LIN {X -0.311,Y -646.142,Z 1277.328,A 0.000,B 0.000,C 90.000,E1 95.049} C_DIS
LIN {X -0.193,Y -640.518,Z 1277.324,A 0.000,B 0.000,C 90.000,E1 94.416} C_DIS
LIN {X 0.051,Y -635.650,Z 1277.322,A 0.000,B 0.000,C 90.000,E1 93.898} C_DIS
LIN {X -0.083,Y -629.590,Z 1277.318,A 0.000,B 0.000,C 90.000,E1 93.326} C_DIS
LIN {X -0.028,Y -623.101,Z 1277.315,A 0.000,B 0.000,C 90.000,E1 92.751} C_DIS
LIN {X 0.105,Y -616.171,Z 1277.312,A 0.000,B 0.000,C 90.000,E1 92.178} C_DIS
LIN {X -0.112,Y -607.322,Z 1277.309,A 0.000,B 0.000,C 90.000,E1 91.547} C_DIS
LIN {X -0.177,Y -601.123,Z 1277.306,A 0.000,B 0.000,C 90.000,E1 91.146} C_DIS
LIN {X 0.025,Y -594.809,Z 1277.304,A 0.000,B 0.000,C 90.000,E1 90.745} C_DIS
LIN {X 0.026,Y -587.877,Z 1277.302,A 0.000,B 0.000,C 90.000,E1 90.401} C_DIS
LIN {X -0.076,Y -580.661,Z 1277.301,A 0.000,B 0.000,C 90.000,E1 90.115} C_DIS
LIN {X 0.222,Y -575.677,Z 1277.300,A 0.000,B 0.000,C 90.000,E1 89.885} C_DIS
LIN {X -0.112,Y -572.688,Z 1277.299,A 0.000,B 0.000,C 90.000,E1 89.771} C_DIS
LIN {X 0.053,Y -572.048,Z 1277.298,A 0.000,B 0.000,C 90.000,E1 89.714} C_DIS
LIN {X -0.053,Y -569.686,Z 1277.297,A 0.000,B 0.000,C 90.000,E1 89.484} C_DIS
LIN {X 0.150,Y -569.196,Z 1277.296,A 0.000,B 0.000,C 90.000,E1 89.312} C_DIS
LIN {X -0.165,Y -568.849,Z 1277.293,A 0.000,B 0.000,C 90.000,E1 88.797} C_DIS
LIN {X -0.001,Y -570.946,Z 1277.278,A 0.000,B 0.000,C 90.000,E1 86.045} C_DIS
LIN {X -0.120,Y -572.846,Z 1277.267,A 0.000,B 0.000,C 90.000,E1 84.147} C_DIS
LIN {X 0.124,Y -574.397,Z 1277.260,A 0.000,B 0.000,C 90.000,E1 82.761} C_DIS
LIN {X 0.031,Y -576.292,Z 1277.251,A 0.000,B 0.000,C 90.000,E1 81.141} C_DIS
LIN {X -0.146,Y -577.751,Z 1277.243,A 0.000,B 0.000,C 90.000,E1 79.803} C_DIS
LIN {X -0.303,Y -578.962,Z 1277.236,A 0.000,B 0.000,C 90.000,E1 78.465} C_DIS
LIN {X 0.237,Y -580.132,Z 1277.228,A 0.000,B 0.000,C 90.000,E1 77.061} C_DIS
LIN {X -0.198,Y -581.224,Z 1277.221,A 0.000,B 0.000,C 90.000,E1 75.755} C_DIS
LIN {X 0.293,Y -581.995,Z 1277.215,A 0.000,B 0.000,C 90.000,E1 74.629} C_DIS
LIN {X 0.231,Y -582.699,Z 1277.209,A 0.000,B 0.000,C 90.000,E1 73.559} C_DIS
LIN {X 0.143,Y -584.243,Z 1277.195,A 0.000,B 0.000,C 90.000,E1 71.148} C_DIS
LIN {X 0.214,Y -585.172,Z 1277.185,A 0.000,B 0.000,C 90.000,E1 69.263} C_DIS
LIN {X -0.156,Y -586.471,Z 1277.173,A 0.000,B 0.000,C 90.000,E1 67.155} C_DIS
LIN {X -0.026,Y -587.736,Z 1277.164,A 0.000,B 0.000,C 90.000,E1 65.537} C_DIS
LIN {X -0.165,Y -588.956,Z 1277.155,A 0.000,B 0.000,C 90.000,E1 63.948} C_DIS
LIN {X -0.113,Y -590.551,Z 1277.145,A 0.000,B 0.000,C 90.000,E1 62.076} C_DIS
LIN {X 0.172,Y -591.848,Z 1277.137,A 0.000,B 0.000,C 90.000,E1 60.717} C_DIS
LIN {X 0.153,Y -593.488,Z 1277.129,A 0.000,B 0.000,C 90.000,E1 59.125} C_DIS
LIN {X 0.262,Y -594.894,Z 1277.121,A 0.000,B 0.000,C 90.000,E1 57.788} C_DIS
LIN {X 0.002,Y -596.798,Z 1277.111,A 0.000,B 0.000,C 90.000,E1 55.960} C_DIS
LIN {X -0.274,Y -598.355,Z 1277.102,A 0.000,B 0.000,C 90.000,E1 54.402} C_DIS
LIN {X 0.327,Y -599.696,Z 1277.093,A 0.000,B 0.000,C 90.000,E1 52.763} C_DIS
LIN {X -0.124,Y -601.169,Z 1277.083,A 0.000,B 0.000,C 90.000,E1 50.964} C_DIS
LIN {X 0.146,Y -601.685,Z 1277.079,A 0.000,B 0.000,C 90.000,E1 50.150} C_DIS
LIN {X -0.038,Y -602.063,Z 1277.074,A 0.000,B 0.000,C 90.000,E1 49.380} C_DIS
LIN {X 0.064,Y -602.737,Z 1277.066,A 0.000,B 0.000,C 90.000,E1 47.796} C_DIS
LIN {X 0.102,Y -603.120,Z 1277.060,A 0.000,B 0.000,C 90.000,E1 46.743} C_DIS
LIN {X -0.264,Y -603.339,Z 1277.054,A 0.000,B 0.000,C 90.000,E1 45.729} C_DIS
LIN {X 0.014,Y -603.317,Z 1277.047,A 0.000,B 0.000,C 90.000,E1 44.393} C_DIS
LIN {X -0.121,Y -603.052,Z 1277.039,A 0.000,B 0.000,C 90.000,E1 43.095} C_DIS
LIN {X 0.160,Y -602.625,Z 1277.032,A 0.000,B 0.000,C 90.000,E1 41.757} C_DIS
LIN {X 0.236,Y -602.215,Z 1277.026,A 0.000,B 0.000,C 90.000,E1 40.701} C_DIS
LIN {X 0.306,Y -601.680,Z 1277.021,A 0.000,B 0.000,C 90.000,E1 39.644} C_DIS
LIN {X -0.262,Y -601.275,Z 1277.016,A 0.000,B 0.000,C 90.000,E1 38.910} C_DIS
LIN {X 0.259,Y -600.534,Z 1277.010,A 0.000,B 0.000,C 90.000,E1 37.810} C_DIS
LIN {X 0.157,Y -599.777,Z 1277.006,A 0.000,B 0.000,C 90.000,E1 37.030} C_DIS
LIN {X 0.048,Y -598.125,Z 1276.999,A 0.000,B 0.000,C 90.000,E1 35.724} C_DIS
LIN {X -0.081,Y -596.974,Z 1276.994,A 0.000,B 0.000,C 90.000,E1 34.945} C_DIS
LIN {X 0.160,Y -595.065,Z 1276.988,A 0.000,B 0.000,C 90.000,E1 33.865} C_DIS
LIN {X -0.003,Y -593.584,Z 1276.984,A 0.000,B 0.000,C 90.000,E1 33.086} C_DIS
LIN {X 0.196,Y -590.897,Z 1276.978,A 0.000,B 0.000,C 90.000,E1 32.005} C_DIS
LIN {X 0.168,Y -588.726,Z 1276.974,A 0.000,B 0.000,C 90.000,E1 31.209} C_DIS
LIN {X 0.121,Y -586.110,Z 1276.969,A 0.000,B 0.000,C 90.000,E1 30.413} C_DIS
LIN {X 0.173,Y -584.179,Z 1276.966,A 0.000,B 0.000,C 90.000,E1 29.873} C_DIS
LIN {X 0.207,Y -581.993,Z 1276.963,A 0.000,B 0.000,C 90.000,E1 29.333} C_DIS
LIN {X 0.011,Y -577.776,Z 1276.958,A 0.000,B 0.000,C 90.000,E1 28.409} C_DIS
LIN {X -0.208,Y -575.700,Z 1276.956,A 0.000,B 0.000,C 90.000,E1 28.025} C_DIS
LIN {X 0.018,Y -570.604,Z 1276.950,A 0.000,B 0.000,C 90.000,E1 27.052} C_DIS
LIN {X 0.012,Y -565.575,Z 1276.946,A 0.000,B 0.000,C 90.000,E1 26.232} C_DIS
LIN {X 0.150,Y -562.014,Z 1276.943,A 0.000,B 0.000,C 90.000,E1 25.668} C_DIS
LIN {X -0.240,Y -558.197,Z 1276.940,A 0.000,B 0.000,C 90.000,E1 25.155} C_DIS
LIN {X -0.150,Y -554.156,Z 1276.937,A 0.000,B 0.000,C 90.000,E1 24.591} C_DIS
LIN {X -0.202,Y -548.717,Z 1276.933,A 0.000,B 0.000,C 90.000,E1 23.898} C_DIS
LIN {X -0.233,Y -541.795,Z 1276.928,A 0.000,B 0.000,C 90.000,E1 23.078} C_DIS
LIN {X 0.234,Y -536.783,Z 1276.925,A 0.000,B 0.000,C 90.000,E1 22.461} C_DIS
LIN {X 0.008,Y -529.038,Z 1276.920,A 0.000,B 0.000,C 90.000,E1 21.642} C_DIS
LIN {X 0.168,Y -521.094,Z 1276.916,A 0.000,B 0.000,C 90.000,E1 20.791} C_DIS
LIN {X 0.048,Y -514.520,Z 1276.912,A 0.000,B 0.000,C 90.000,E1 20.120} C_DIS
LIN {X 0.049,Y -503.625,Z 1276.906,A 0.000,B 0.000,C 90.000,E1 19.033} C_DIS
LIN {X 0.099,Y -491.041,Z 1276.899,A 0.000,B 0.000,C 90.000,E1 17.819} C_DIS
LIN {X 0.101,Y -485.191,Z 1276.896,A 0.000,B 0.000,C 90.000,E1 17.275} C_DIS
LIN {X 0.041,Y -476.407,Z 1276.892,A 0.000,B 0.000,C 90.000,E1 16.496} C_DIS
LIN {X -0.223,Y -466.089,Z 1276.887,A 0.000,B 0.000,C 90.000,E1 15.607} C_DIS
LIN {X 0.108,Y -448.357,Z 1276.878,A 0.000,B 0.000,C 90.000,E1 13.953} C_DIS
LIN {X 0.113,Y -425.103,Z 1276.865,A 0.000,B 0.000,C 90.000,E1 11.658} C_DIS
LIN {X 0.141,Y -409.302,Z 1276.855,A 0.000,B 0.000,C 90.000,E1 9.962} C_DIS
LIN {X 0.139,Y -399.520,Z 1276.849,A 0.000,B 0.000,C 90.000,E1 8.859} C_DIS
LIN {X -0.160,Y -395.627,Z 1276.846,A 0.000,B 0.000,C 90.000,E1 8.341} C_DIS
LIN {X 0.010,Y -394.992,Z 1276.845,A 0.000,B 0.000,C 90.000,E1 8.163} C_DIS
LIN {X -0.028,Y -394.987,Z 1276.845,A 0.000,B 0.000,C 90.000,E1 8.163} C_DIS
LIN {X -0.121,Y -395.323,Z 1276.845,A 0.000,B 0.000,C 90.000,E1 8.049} C_DIS
LIN {X 0.042,Y -396.381,Z 1276.844,A 0.000,B 0.000,C 90.000,E1 7.871} C_DIS
LIN {X -0.132,Y -399.602,Z 1276.842,A 0.000,B 0.000,C 90.000,E1 7.587} C_DIS
LIN {X -0.017,Y -402.154,Z 1276.841,A 0.000,B 0.000,C 90.000,E1 7.409} C_DIS
LIN {X 0.161,Y -410.548,Z 1276.839,A 0.000,B 0.000,C 90.000,E1 6.891} C_DIS
LIN {X 0.052,Y -417.083,Z 1276.836,A 0.000,B 0.000,C 90.000,E1 6.486} C_DIS
LIN {X 0.081,Y -424.986,Z 1276.833,A 0.000,B 0.000,C 90.000,E1 5.910} C_DIS
LIN {X -0.203,Y -432.931,Z 1276.830,A 0.000,B 0.000,C 90.000,E1 5.334} C_DIS
LIN {X 0.214,Y -442.339,Z 1276.825,A 0.000,B 0.000,C 90.000,E1 4.531} C_DIS
LIN {X -0.008,Y -453.087,Z 1276.820,A 0.000,B 0.000,C 90.000,E1 3.669} C_DIS
LIN {X -0.188,Y -460.478,Z 1276.817,A 0.000,B 0.000,C 90.000,E1 3.037} C_DIS
LIN {X -0.215,Y -467.568,Z 1276.813,A 0.000,B 0.000,C 90.000,E1 2.350} C_DIS
LIN {X 0.238,Y -473.173,Z 1276.810,A 0.000,B 0.000,C 90.000,E1 1.718} C_DIS
LIN {X -0.175,Y -479.787,Z 1276.806,A 0.000,B 0.000,C 90.000,E1 1.031} C_DIS
LIN {X 0.132,Y -486.135,Z 1276.801,A 0.000,B 0.000,C 90.000,E1 0.229} C_DIS
LIN {X 0.020,Y -491.932,Z 1276.797,A 0.000,B 0.000,C 90.000,E1 359.484} C_DIS
LIN {X 0.069,Y -498.184,Z 1276.792,A 0.000,B 0.000,C 90.000,E1 358.568} C_DIS
LIN {X 0.012,Y -503.008,Z 1276.788,A 0.000,B 0.000,C 90.000,E1 357.822} C_DIS
LIN {X -0.021,Y -507.526,Z 1276.784,A 0.000,B 0.000,C 90.000,E1 357.078} C_DIS
LIN {X -0.196,Y -510.965,Z 1276.781,A 0.000,B 0.000,C 90.000,E1 356.502} C_DIS
LIN {X -0.128,Y -514.957,Z 1276.776,A 0.000,B 0.000,C 90.000,E1 355.755} C_DIS
LIN {X 0.272,Y -517.958,Z 1276.773,A 0.000,B 0.000,C 90.000,E1 355.122} C_DIS
LIN {X 0.111,Y -523.509,Z 1276.767,A 0.000,B 0.000,C 90.000,E1 353.970} C_DIS
LIN {X -0.230,Y -526.640,Z 1276.763,A 0.000,B 0.000,C 90.000,E1 353.280} C_DIS
LIN {X -0.245,Y -530.008,Z 1276.758,A 0.000,B 0.000,C 90.000,E1 352.413} C_DIS
LIN {X -0.224,Y -533.177,Z 1276.753,A 0.000,B 0.000,C 90.000,E1 351.546} C_DIS
LIN {X -0.173,Y -536.035,Z 1276.748,A 0.000,B 0.000,C 90.000,E1 350.679} C_DIS
LIN {X -0.001,Y -538.590,Z 1276.743,A 0.000,B 0.000,C 90.000,E1 349.803} C_DIS
LIN {X 0.280,Y -541.711,Z 1276.737,A 0.000,B 0.000,C 90.000,E1 348.634} C_DIS
LIN {X 0.163,Y -545.005,Z 1276.729,A 0.000,B 0.000,C 90.000,E1 347.229} C_DIS
LIN {X -0.096,Y -546.798,Z 1276.724,A 0.000,B 0.000,C 90.000,E1 346.408} C_DIS
LIN {X -0.206,Y -548.326,Z 1276.720,A 0.000,B 0.000,C 90.000,E1 345.574} C_DIS
LIN {X 0.091,Y -549.695,Z 1276.715,A 0.000,B 0.000,C 90.000,E1 344.700} C_DIS
LIN {X 0.267,Y -551.225,Z 1276.709,A 0.000,B 0.000,C 90.000,E1 343.559} C_DIS
LIN {X -0.221,Y -552.400,Z 1276.703,A 0.000,B 0.000,C 90.000,E1 342.489} C_DIS
LIN {X 0.171,Y -553.178,Z 1276.696,A 0.000,B 0.000,C 90.000,E1 341.329} C_DIS
LIN {X 0.119,Y -553.406,Z 1276.692,A 0.000,B 0.000,C 90.000,E1 340.496} C_DIS
LIN {X -0.271,Y -553.242,Z 1276.687,A 0.000,B 0.000,C 90.000,E1 339.699} C_DIS
LIN {X -0.145,Y -552.772,Z 1276.682,A 0.000,B 0.000,C 90.000,E1 338.847} C_DIS
LIN {X 0.177,Y -552.087,Z 1276.678,A 0.000,B 0.000,C 90.000,E1 337.975} C_DIS
LIN {X 0.045,Y -550.521,Z 1276.672,A 0.000,B 0.000,C 90.000,E1 336.869} C_DIS
LIN {X 0.077,Y -549.566,Z 1276.668,A 0.000,B 0.000,C 90.000,E1 336.305} C_DIS
LIN {X 0.120,Y -547.475,Z 1276.662,A 0.000,B 0.000,C 90.000,E1 335.177} C_DIS
LIN {X -0.121,Y -546.881,Z 1276.661,A 0.000,B 0.000,C 90.000,E1 334.921} C_DIS
LIN {X -0.126,Y -544.680,Z 1276.656,A 0.000,B 0.000,C 90.000,E1 334.076} C_DIS
LIN {X 0.097,Y -542.293,Z 1276.651,A 0.000,B 0.000,C 90.000,E1 333.204} C_DIS
LIN {X 0.049,Y -539.456,Z 1276.646,A 0.000,B 0.000,C 90.000,E1 332.359} C_DIS
LIN {X -0.027,Y -536.198,Z 1276.642,A 0.000,B 0.000,C 90.000,E1 331.513} C_DIS
LIN {X 0.004,Y -533.130,Z 1276.638,A 0.000,B 0.000,C 90.000,E1 330.795} C_DIS
LIN {X 0.003,Y -529.676,Z 1276.634,A 0.000,B 0.000,C 90.000,E1 330.078} C_DIS
LIN {X 0.120,Y -526.538,Z 1276.631,A 0.000,B 0.000,C 90.000,E1 329.488} C_DIS
LIN {X -0.067,Y -518.976,Z 1276.623,A 0.000,B 0.000,C 90.000,E1 328.201} C_DIS
LIN {X 0.342,Y -511.317,Z 1276.616,A 0.000,B 0.000,C 90.000,E1 326.834} C_DIS
LIN {X 0.069,Y -507.847,Z 1276.612,A 0.000,B 0.000,C 90.000,E1 326.167} C_DIS
LIN {X 0.066,Y -505.793,Z 1276.610,A 0.000,B 0.000,C 90.000,E1 325.722} C_DIS
LIN {X 0.275,Y -503.558,Z 1276.606,A 0.000,B 0.000,C 90.000,E1 325.102} C_DIS
LIN {X -0.055,Y -501.327,Z 1276.601,A 0.000,B 0.000,C 90.000,E1 324.242} C_DIS
LIN {X -0.003,Y -499.802,Z 1276.596,A 0.000,B 0.000,C 90.000,E1 323.336} C_DIS
LIN {X 0.204,Y -498.853,Z 1276.590,A 0.000,B 0.000,C 90.000,E1 322.110} C_DIS
LIN {X -0.256,Y -498.480,Z 1276.580,A 0.000,B 0.000,C 90.000,E1 320.356} C_DIS
LIN {X -0.273,Y -498.662,Z 1276.571,A 0.000,B 0.000,C 90.000,E1 318.852} C_DIS
LIN {X -0.101,Y -498.971,Z 1276.561,A 0.000,B 0.000,C 90.000,E1 317.025} C_DIS
LIN {X 0.195,Y -499.188,Z 1276.553,A 0.000,B 0.000,C 90.000,E1 315.486} C_DIS
LIN {X -0.205,Y -499.520,Z 1276.545,A 0.000,B 0.000,C 90.000,E1 314.028} C_DIS
LIN {X -0.177,Y -499.919,Z 1276.533,A 0.000,B 0.000,C 90.000,E1 311.919} C_DIS
LIN {X 0.158,Y -500.203,Z 1276.524,A 0.000,B 0.000,C 90.000,E1 310.378} C_DIS
LIN {X -0.084,Y -500.475,Z 1276.513,A 0.000,B 0.000,C 90.000,E1 308.302} C_DIS
LIN {X 0.129,Y -500.611,Z 1276.506,A 0.000,B 0.000,C 90.000,E1 307.076} C_DIS
LIN {X -0.193,Y -500.797,Z 1276.496,A 0.000,B 0.000,C 90.000,E1 305.311} C_DIS
LIN {X -0.148,Y -500.762,Z 1276.491,A 0.000,B 0.000,C 90.000,E1 304.405} C_DIS
LIN {X 0.021,Y -500.577,Z 1276.488,A 0.000,B 0.000,C 90.000,E1 303.785} C_DIS
LIN {X 0.061,Y -499.962,Z 1276.483,A 0.000,B 0.000,C 90.000,E1 302.880} C_DIS
LIN {X -0.178,Y -498.986,Z 1276.478,A 0.000,B 0.000,C 90.000,E1 302.005} C_DIS
LIN {X -0.027,Y -498.060,Z 1276.474,A 0.000,B 0.000,C 90.000,E1 301.386} C_DIS
LIN {X 0.002,Y -497.411,Z 1276.473,A 0.000,B 0.000,C 90.000,E1 301.082} C_DIS
LIN {X -0.140,Y -496.590,Z 1276.471,A 0.000,B 0.000,C 90.000,E1 300.797} C_DIS
LIN {X 0.140,Y -495.401,Z 1276.469,A 0.000,B 0.000,C 90.000,E1 300.463} C_DIS
LIN {X -0.078,Y -481.481,Z 1276.453,A 0.000,B 0.000,C 90.000,E1 297.590} C_DIS
LIN {X -0.130,Y -469.289,Z 1276.437,A 0.000,B 0.000,C 90.000,E1 294.643} C_DIS
LIN {X 0.033,Y -458.237,Z 1276.419,A 0.000,B 0.000,C 90.000,E1 291.461} C_DIS
LIN {X -0.127,Y -448.080,Z 1276.400,A 0.000,B 0.000,C 90.000,E1 287.946} C_DIS
LIN {X 0.040,Y -439.286,Z 1276.378,A 0.000,B 0.000,C 90.000,E1 284.008} C_DIS
LIN {X 0.059,Y -431.922,Z 1276.352,A 0.000,B 0.000,C 90.000,E1 279.378} C_DIS
LIN {X -0.009,Y -426.740,Z 1276.317,A 0.000,B 0.000,C 90.000,E1 273.037} C_DIS
LIN {X -0.072,Y -429.939,Z 1276.259,A 0.000,B 0.000,C 90.000,E1 262.648} C_DIS
LIN {X 0.033,Y -436.735,Z 1276.231,A 0.000,B 0.000,C 90.000,E1 257.645} C_DIS
LIN {X 0.143,Y -444.731,Z 1276.209,A 0.000,B 0.000,C 90.000,E1 253.685} C_DIS
LIN {X 0.142,Y -454.140,Z 1276.190,A 0.000,B 0.000,C 90.000,E1 250.115} C_DIS
LIN {X 0.100,Y -464.499,Z 1276.172,A 0.000,B 0.000,C 90.000,E1 246.922} C_DIS
LIN {X 0.029,Y -465.631,Z 1276.170,A 0.000,B 0.000,C 90.000,E1 246.613} C_DIS
LIN {X -0.037,Y -466.547,Z 1276.168,A 0.000,B 0.000,C 90.000,E1 246.305} C_DIS
LIN {X 0.089,Y -467.104,Z 1276.167,A 0.000,B 0.000,C 90.000,E1 245.973} C_DIS
LIN {X -0.028,Y -467.772,Z 1276.163,A 0.000,B 0.000,C 90.000,E1 245.357} C_DIS
LIN {X -0.002,Y -468.158,Z 1276.158,A 0.000,B 0.000,C 90.000,E1 244.409} C_DIS
LIN {X 0.026,Y -468.133,Z 1276.153,A 0.000,B 0.000,C 90.000,E1 243.461} C_DIS
LIN {X -0.152,Y -467.862,Z 1276.147,A 0.000,B 0.000,C 90.000,E1 242.538} C_DIS
LIN {X -0.164,Y -466.746,Z 1276.135,A 0.000,B 0.000,C 90.000,E1 240.333} C_DIS
LIN {X -0.199,Y -466.056,Z 1276.128,A 0.000,B 0.000,C 90.000,E1 239.076} C_DIS
LIN {X -0.107,Y -464.826,Z 1276.118,A 0.000,B 0.000,C 90.000,E1 237.168} C_DIS
LIN {X -0.046,Y -463.576,Z 1276.107,A 0.000,B 0.000,C 90.000,E1 235.261} C_DIS
LIN {X 0.000,Y -462.164,Z 1276.093,A 0.000,B 0.000,C 90.000,E1 232.718} C_DIS
LIN {X -0.194,Y -461.159,Z 1276.081,A 0.000,B 0.000,C 90.000,E1 230.517} C_DIS
LIN {X 0.179,Y -460.402,Z 1276.068,A 0.000,B 0.000,C 90.000,E1 228.243} C_DIS
LIN {X -0.108,Y -459.649,Z 1276.054,A 0.000,B 0.000,C 90.000,E1 225.729} C_DIS
LIN {X 0.101,Y -459.329,Z 1276.045,A 0.000,B 0.000,C 90.000,E1 224.109} C_DIS
LIN {X 0.050,Y -459.570,Z 1276.022,A 0.000,B 0.000,C 90.000,E1 219.967} C_DIS
LIN {X -0.047,Y -461.359,Z 1275.997,A 0.000,B 0.000,C 90.000,E1 215.518} C_DIS
LIN {X 0.109,Y -464.598,Z 1275.978,A 0.000,B 0.000,C 90.000,E1 212.005} C_DIS
LIN {X -0.060,Y -466.897,Z 1275.967,A 0.000,B 0.000,C 90.000,E1 210.129} C_DIS
LIN {X -0.162,Y -468.726,Z 1275.959,A 0.000,B 0.000,C 90.000,E1 208.565} C_DIS
LIN {X -0.009,Y -472.249,Z 1275.943,A 0.000,B 0.000,C 90.000,E1 205.720} C_DIS
LIN {X 0.107,Y -475.892,Z 1275.929,A 0.000,B 0.000,C 90.000,E1 203.206} C_DIS
LIN {X -0.031,Y -479.891,Z 1275.915,A 0.000,B 0.000,C 90.000,E1 200.737} C_DIS
LIN {X 0.227,Y -484.176,Z 1275.901,A 0.000,B 0.000,C 90.000,E1 198.236} C_DIS
LIN {X -0.176,Y -488.111,Z 1275.890,A 0.000,B 0.000,C 90.000,E1 196.134} C_DIS
LIN {X -0.164,Y -491.495,Z 1275.879,A 0.000,B 0.000,C 90.000,E1 194.300} C_DIS
LIN {X -0.184,Y -494.974,Z 1275.869,A 0.000,B 0.000,C 90.000,E1 192.479} C_DIS
LIN {X 0.042,Y -497.397,Z 1275.863,A 0.000,B 0.000,C 90.000,E1 191.243} C_DIS
LIN {X -0.109,Y -501.457,Z 1275.851,A 0.000,B 0.000,C 90.000,E1 189.151} C_DIS
LIN {X -0.224,Y -505.709,Z 1275.839,A 0.000,B 0.000,C 90.000,E1 187.068} C_DIS
LIN {X -0.133,Y -508.582,Z 1275.831,A 0.000,B 0.000,C 90.000,E1 185.568} C_DIS
LIN {X -0.180,Y -512.592,Z 1275.819,A 0.000,B 0.000,C 90.000,E1 183.498} C_DIS
LIN {X -0.039,Y -515.339,Z 1275.811,A 0.000,B 0.000,C 90.000,E1 182.007} C_DIS
LIN {X 0.152,Y -517.962,Z 1275.803,A 0.000,B 0.000,C 90.000,E1 180.516} C_DIS
LIN {X -0.194,Y -520.978,Z 1275.793,A 0.000,B 0.000,C 90.000,E1 178.797} C_DIS
LIN {X 0.098,Y -523.264,Z 1275.785,A 0.000,B 0.000,C 90.000,E1 177.306} C_DIS
LIN {X -0.052,Y -524.913,Z 1275.779,A 0.000,B 0.000,C 90.000,E1 176.159} C_DIS
LIN {X -0.140,Y -526.368,Z 1275.772,A 0.000,B 0.000,C 90.000,E1 175.008} C_DIS
LIN {X -0.245,Y -527.935,Z 1275.764,A 0.000,B 0.000,C 90.000,E1 173.571} C_DIS
LIN {X -0.207,Y -528.448,Z 1275.761,A 0.000,B 0.000,C 90.000,E1 172.989} C_DIS
LIN {X -0.245,Y -529.354,Z 1275.755,A 0.000,B 0.000,C 90.000,E1 171.837} C_DIS
LIN {X -0.236,Y -529.859,Z 1275.750,A 0.000,B 0.000,C 90.000,E1 170.971} C_DIS
LIN {X -0.099,Y -530.288,Z 1275.743,A 0.000,B 0.000,C 90.000,E1 169.803} C_DIS
LIN {X 0.013,Y -530.471,Z 1275.739,A 0.000,B 0.000,C 90.000,E1 168.926} C_DIS
LIN {X 0.167,Y -530.629,Z 1275.732,A 0.000,B 0.000,C 90.000,E1 167.757} C_DIS
LIN {X -0.201,Y -530.427,Z 1275.726,A 0.000,B 0.000,C 90.000,E1 166.645} C_DIS
LIN {X -0.219,Y -529.994,Z 1275.714,A 0.000,B 0.000,C 90.000,E1 164.629} C_DIS
LIN {X -0.278,Y -529.654,Z 1275.705,A 0.000,B 0.000,C 90.000,E1 162.906} C_DIS
LIN {X 0.096,Y -529.738,Z 1275.700,A 0.000,B 0.000,C 90.000,E1 162.000} C_DIS
LIN {X -0.016,Y -530.007,Z 1275.694,A 0.000,B 0.000,C 90.000,E1 160.859} C_DIS
LIN {X 0.047,Y -530.830,Z 1275.687,A 0.000,B 0.000,C 90.000,E1 159.699} C_DIS
LIN {X 0.124,Y -532.438,Z 1275.681,A 0.000,B 0.000,C 90.000,E1 158.539} C_DIS
LIN {X 0.022,Y -533.543,Z 1275.678,A 0.000,B 0.000,C 90.000,E1 157.975} C_DIS
LIN {X -0.150,Y -536.632,Z 1275.671,A 0.000,B 0.000,C 90.000,E1 156.847} C_DIS
LIN {X -0.136,Y -540.491,Z 1275.666,A 0.000,B 0.000,C 90.000,E1 155.845} C_DIS
LIN {X 0.188,Y -543.912,Z 1275.662,A 0.000,B 0.000,C 90.000,E1 155.101} C_DIS
LIN {X 0.050,Y -548.091,Z 1275.658,A 0.000,B 0.000,C 90.000,E1 154.409} C_DIS
LIN {X 0.074,Y -553.835,Z 1275.653,A 0.000,B 0.000,C 90.000,E1 153.563} C_DIS
LIN {X -0.006,Y -562.191,Z 1275.647,A 0.000,B 0.000,C 90.000,E1 152.487} C_DIS
LIN {X 0.194,Y -572.757,Z 1275.641,A 0.000,B 0.000,C 90.000,E1 151.257} C_DIS
LIN {X 0.034,Y -580.993,Z 1275.635,A 0.000,B 0.000,C 90.000,E1 150.333} C_DIS
LIN {X -0.147,Y -589.113,Z 1275.630,A 0.000,B 0.000,C 90.000,E1 149.410} C_DIS
LIN {X 0.195,Y -593.388,Z 1275.627,A 0.000,B 0.000,C 90.000,E1 148.869} C_DIS
LIN {X 0.037,Y -596.482,Z 1275.625,A 0.000,B 0.000,C 90.000,E1 148.486} C_DIS
LIN {X -0.350,Y -600.834,Z 1275.622,A 0.000,B 0.000,C 90.000,E1 147.995} C_DIS
LIN {X -0.157,Y -605.737,Z 1275.618,A 0.000,B 0.000,C 90.000,E1 147.327} C_DIS
LIN {X 0.030,Y -609.497,Z 1275.616,A 0.000,B 0.000,C 90.000,E1 146.786} C_DIS
LIN {X -0.267,Y -613.125,Z 1275.613,A 0.000,B 0.000,C 90.000,E1 146.294} C_DIS
LIN {X 0.034,Y -615.755,Z 1275.610,A 0.000,B 0.000,C 90.000,E1 145.881} C_DIS
LIN {X -0.241,Y -619.719,Z 1275.607,A 0.000,B 0.000,C 90.000,E1 145.261} C_DIS
LIN {X -0.126,Y -623.490,Z 1275.603,A 0.000,B 0.000,C 90.000,E1 144.609} C_DIS
LIN {X 0.193,Y -625.625,Z 1275.601,A 0.000,B 0.000,C 90.000,E1 144.196} C_DIS
LIN {X -0.157,Y -630.282,Z 1275.596,A 0.000,B 0.000,C 90.000,E1 143.336} C_DIS
LIN {X -0.090,Y -635.452,Z 1275.590,A 0.000,B 0.000,C 90.000,E1 142.190} C_DIS
LIN {X 0.051,Y -639.559,Z 1275.584,A 0.000,B 0.000,C 90.000,E1 141.170} C_DIS
LIN {X 0.154,Y -644.133,Z 1275.577,A 0.000,B 0.000,C 90.000,E1 139.908} C_DIS
LIN {X -0.161,Y -648.283,Z 1275.570,A 0.000,B 0.000,C 90.000,E1 138.690} C_DIS
LIN {X 0.081,Y -651.540,Z 1275.565,A 0.000,B 0.000,C 90.000,E1 137.676} C_DIS
LIN {X -0.077,Y -654.541,Z 1275.559,A 0.000,B 0.000,C 90.000,E1 136.701} C_DIS
LIN {X -0.315,Y -659.847,Z 1275.550,A 0.000,B 0.000,C 90.000,E1 135.000} C_DIS
LIN {X 0.052,Y -665.376,Z 1275.540,A 0.000,B 0.000,C 90.000,E1 133.257} C_DIS
LIN {X 0.037,Y -669.248,Z 1275.534,A 0.000,B 0.000,C 90.000,E1 132.043} C_DIS
LIN {X 0.114,Y -672.295,Z 1275.528,A 0.000,B 0.000,C 90.000,E1 131.067} C_DIS
LIN {X -0.182,Y -675.999,Z 1275.522,A 0.000,B 0.000,C 90.000,E1 129.886} C_DIS
LIN {X 0.012,Y -679.496,Z 1275.515,A 0.000,B 0.000,C 90.000,E1 128.669} C_DIS
LIN {X -0.202,Y -682.196,Z 1275.510,A 0.000,B 0.000,C 90.000,E1 127.729} C_DIS
LIN {X 0.194,Y -685.413,Z 1275.503,A 0.000,B 0.000,C 90.000,E1 126.503} C_DIS
LIN {X -0.132,Y -688.896,Z 1275.495,A 0.000,B 0.000,C 90.000,E1 125.105} C_DIS
LIN {X 0.327,Y -691.077,Z 1275.490,A 0.000,B 0.000,C 90.000,E1 124.119} C_DIS
LIN {X 0.073,Y -693.468,Z 1275.483,A 0.000,B 0.000,C 90.000,E1 122.959} C_DIS
LIN {X -0.145,Y -695.723,Z 1275.477,A 0.000,B 0.000,C 90.000,E1 121.799} C_DIS
LIN {X -0.001,Y -696.961,Z 1275.473,A 0.000,B 0.000,C 90.000,E1 121.082} C_DIS
LIN {X 0.170,Y -698.515,Z 1275.468,A 0.000,B 0.000,C 90.000,E1 120.129} C_DIS
LIN {X 0.269,Y -700.207,Z 1275.461,A 0.000,B 0.000,C 90.000,E1 118.949} C_DIS
LIN {X 0.121,Y -701.311,Z 1275.456,A 0.000,B 0.000,C 90.000,E1 118.025} C_DIS
LIN {X 0.001,Y -701.994,Z 1275.452,A 0.000,B 0.000,C 90.000,E1 117.334} C_DIS
LIN {X -0.068,Y -702.330,Z 1275.449,A 0.000,B 0.000,C 90.000,E1 116.873} C_DIS
LIN {X 0.141,Y -702.484,Z 1275.445,A 0.000,B 0.000,C 90.000,E1 116.155} C_DIS
LIN {X -0.239,Y -702.457,Z 1275.443,A 0.000,B 0.000,C 90.000,E1 115.720} C_DIS
LIN {X 0.319,Y -702.253,Z 1275.440,A 0.000,B 0.000,C 90.000,E1 115.207} C_DIS
LIN {X -0.059,Y -701.883,Z 1275.438,A 0.000,B 0.000,C 90.000,E1 114.771} C_DIS
LIN {X -0.435,Y -701.208,Z 1275.435,A 0.000,B 0.000,C 90.000,E1 114.335} C_DIS
LIN {X -0.160,Y -700.780,Z 1275.434,A 0.000,B 0.000,C 90.000,E1 114.079} C_DIS
LIN {X 0.233,Y -698.474,Z 1275.431,A 0.000,B 0.000,C 90.000,E1 113.462} C_DIS
LIN {X -0.275,Y -697.726,Z 1275.430,A 0.000,B 0.000,C 90.000,E1 113.387} C_DIS
LIN {X -0.266,Y -694.256,Z 1275.427,A 0.000,B 0.000,C 90.000,E1 112.950} C_DIS
LIN {X -0.141,Y -693.113,Z 1275.427,A 0.000,B 0.000,C 90.000,E1 112.823} C_DIS
LIN {X -0.018,Y -691.351,Z 1275.426,A 0.000,B 0.000,C 90.000,E1 112.695} C_DIS
LIN {X 0.102,Y -689.316,Z 1275.426,A 0.000,B 0.000,C 90.000,E1 112.589} C_DIS
LIN {X -0.167,Y -683.742,Z 1275.424,A 0.000,B 0.000,C 90.000,E1 112.386} C_DIS
LIN {X -0.355,Y -681.829,Z 1275.424,A 0.000,B 0.000,C 90.000,E1 112.333} C_DIS
LIN {X 0.345,Y -679.470,Z 1275.424,A 0.000,B 0.000,C 90.000,E1 112.206} C_DIS
LIN {X -0.256,Y -676.343,Z 1275.423,A 0.000,B 0.000,C 90.000,E1 112.206} C_DIS
LIN {X 0.189,Y -669.684,Z 1275.423,A 0.000,B 0.000,C 90.000,E1 112.099} C_DIS
LIN {X 0.121,Y -637.201,Z 1275.423,A 0.000,B 0.000,C 90.000,E1 112.099} C_DIS
LIN {X -0.143,Y -634.444,Z 1275.422,A 0.000,B 0.000,C 90.000,E1 112.025} C_DIS
LIN {X -0.185,Y -634.372,Z 1275.422,A 0.000,B 0.000,C 90.000,E1 112.025} C_DIS
LIN {X -0.226,Y -634.350,Z 1275.422,A 0.000,B 0.000,C 90.000,E1 112.025} C_DIS
LIN {X -0.268,Y -634.353,Z 1275.422,A 0.000,B 0.000,C 90.000,E1 112.025} C_DIS
LIN {X 0.000,Y -634.744,Z 1275.421,A 0.000,B 0.000,C 90.000,E1 111.844} C_DIS
LIN {X 0.016,Y -635.197,Z 1275.421,A 0.000,B 0.000,C 90.000,E1 111.716} C_DIS
LIN {X -0.130,Y -636.710,Z 1275.419,A 0.000,B 0.000,C 90.000,E1 111.461} C_DIS
LIN {X 0.282,Y -644.750,Z 1275.413,A 0.000,B 0.000,C 90.000,E1 110.301} C_DIS
LIN {X -0.005,Y -648.778,Z 1275.410,A 0.000,B 0.000,C 90.000,E1 109.704} C_DIS
LIN {X -0.180,Y -653.537,Z 1275.405,A 0.000,B 0.000,C 90.000,E1 108.852} C_DIS
LIN {X -0.143,Y -657.164,Z 1275.401,A 0.000,B 0.000,C 90.000,E1 108.109} C_DIS
LIN {X 0.141,Y -660.483,Z 1275.396,A 0.000,B 0.000,C 90.000,E1 107.347} C_DIS
LIN {X 0.032,Y -663.525,Z 1275.392,A 0.000,B 0.000,C 90.000,E1 106.622} C_DIS
LIN {X -0.054,Y -666.201,Z 1275.388,A 0.000,B 0.000,C 90.000,E1 105.898} C_DIS
LIN {X -0.298,Y -668.380,Z 1275.384,A 0.000,B 0.000,C 90.000,E1 105.190} C_DIS
LIN {X 0.129,Y -670.158,Z 1275.380,A 0.000,B 0.000,C 90.000,E1 104.426} C_DIS
LIN {X 0.089,Y -671.392,Z 1275.376,A 0.000,B 0.000,C 90.000,E1 103.703} C_DIS
LIN {X -0.196,Y -672.041,Z 1275.374,A 0.000,B 0.000,C 90.000,E1 103.244} C_DIS
LIN {X 0.275,Y -672.524,Z 1275.370,A 0.000,B 0.000,C 90.000,E1 102.479} C_DIS
LIN {X 0.152,Y -672.660,Z 1275.367,A 0.000,B 0.000,C 90.000,E1 102.007} C_DIS
LIN {X -0.035,Y -672.430,Z 1275.363,A 0.000,B 0.000,C 90.000,E1 101.299} C_DIS
LIN {X -0.293,Y -672.037,Z 1275.360,A 0.000,B 0.000,C 90.000,E1 100.838} C_DIS
LIN {X 0.235,Y -671.447,Z 1275.357,A 0.000,B 0.000,C 90.000,E1 100.310} C_DIS
LIN {X -0.022,Y -670.578,Z 1275.355,A 0.000,B 0.000,C 90.000,E1 99.849} C_DIS
LIN {X -0.169,Y -669.511,Z 1275.352,A 0.000,B 0.000,C 90.000,E1 99.378} C_DIS
LIN {X 0.226,Y -668.076,Z 1275.349,A 0.000,B 0.000,C 90.000,E1 98.859} C_DIS
LIN {X -0.134,Y -665.290,Z 1275.345,A 0.000,B 0.000,C 90.000,E1 98.163} C_DIS
LIN {X 0.238,Y -663.087,Z 1275.343,A 0.000,B 0.000,C 90.000,E1 97.644} C_DIS
LIN {X -0.158,Y -659.768,Z 1275.339,A 0.000,B 0.000,C 90.000,E1 97.068} C_DIS
LIN {X 0.177,Y -656.786,Z 1275.337,A 0.000,B 0.000,C 90.000,E1 96.549} C_DIS
LIN {X -0.197,Y -652.580,Z 1275.333,A 0.000,B 0.000,C 90.000,E1 95.967} C_DIS
LIN {X -0.029,Y -647.785,Z 1275.330,A 0.000,B 0.000,C 90.000,E1 95.334} C_DIS
LIN {X 0.160,Y -643.549,Z 1275.327,A 0.000,B 0.000,C 90.000,E1 94.821} C_DIS
LIN {X -0.260,Y -638.941,Z 1275.324,A 0.000,B 0.000,C 90.000,E1 94.359} C_DIS
LIN {X -0.014,Y -633.949,Z 1275.321,A 0.000,B 0.000,C 90.000,E1 93.841} C_DIS
LIN {X -0.140,Y -629.079,Z 1275.319,A 0.000,B 0.000,C 90.000,E1 93.383} C_DIS
LIN {X -0.227,Y -622.346,Z 1275.316,A 0.000,B 0.000,C 90.000,E1 92.808} C_DIS
LIN {X -0.133,Y -615.240,Z 1275.312,A 0.000,B 0.000,C 90.000,E1 92.236} C_DIS
LIN {X 0.256,Y -607.938,Z 1275.309,A 0.000,B 0.000,C 90.000,E1 91.661} C_DIS
LIN {X 0.122,Y -601.831,Z 1275.307,A 0.000,B 0.000,C 90.000,E1 91.260} C_DIS
LIN {X 0.281,Y -595.531,Z 1275.305,A 0.000,B 0.000,C 90.000,E1 90.859} C_DIS
LIN {X -0.189,Y -590.267,Z 1275.303,A 0.000,B 0.000,C 90.000,E1 90.630} C_DIS
LIN {X 0.245,Y -584.841,Z 1275.302,A 0.000,B 0.000,C 90.000,E1 90.344} C_DIS
LIN {X 0.200,Y -576.109,Z 1275.300,A 0.000,B 0.000,C 90.000,E1 90.000} C_DIS
LIN {X 0.074,Y -572.307,Z 1275.299,A 0.000,B 0.000,C 90.000,E1 89.828} C_DIS
LIN {X 0.037,Y -569.501,Z 1275.297,A 0.000,B 0.000,C 90.000,E1 89.542} C_DIS
LIN {X -0.003,Y -569.475,Z 1275.297,A 0.000,B 0.000,C 90.000,E1 89.542} C_DIS
LIN {X -0.149,Y -568.956,Z 1275.297,A 0.000,B 0.000,C 90.000,E1 89.370} C_DIS
LIN {X -0.069,Y -568.773,Z 1275.295,A 0.000,B 0.000,C 90.000,E1 89.083} C_DIS
LIN {X 0.057,Y -568.746,Z 1275.293,A 0.000,B 0.000,C 90.000,E1 88.797} C_DIS
LIN {X -0.033,Y -570.368,Z 1275.281,A 0.000,B 0.000,C 90.000,E1 86.617} C_DIS
LIN {X -0.027,Y -572.503,Z 1275.269,A 0.000,B 0.000,C 90.000,E1 84.432} C_DIS
LIN {X -0.228,Y -574.330,Z 1275.260,A 0.000,B 0.000,C 90.000,E1 82.818} C_DIS
LIN {X -0.115,Y -576.500,Z 1275.250,A 0.000,B 0.000,C 90.000,E1 80.905} C_DIS
LIN {X 0.069,Y -577.645,Z 1275.243,A 0.000,B 0.000,C 90.000,E1 79.803} C_DIS
LIN {X -0.089,Y -578.854,Z 1275.236,A 0.000,B 0.000,C 90.000,E1 78.465} C_DIS
LIN {X -0.116,Y -580.002,Z 1275.228,A 0.000,B 0.000,C 90.000,E1 77.117} C_DIS
LIN {X -0.213,Y -580.889,Z 1275.222,A 0.000,B 0.000,C 90.000,E1 76.047} C_DIS
LIN {X -0.061,Y -581.848,Z 1275.215,A 0.000,B 0.000,C 90.000,E1 74.685} C_DIS
LIN {X -0.121,Y -582.536,Z 1275.209,A 0.000,B 0.000,C 90.000,E1 73.614} C_DIS
LIN {X 0.157,Y -584.076,Z 1275.196,A 0.000,B 0.000,C 90.000,E1 71.167} C_DIS
LIN {X -0.136,Y -585.007,Z 1275.185,A 0.000,B 0.000,C 90.000,E1 69.316} C_DIS
LIN {X -0.191,Y -586.313,Z 1275.173,A 0.000,B 0.000,C 90.000,E1 67.177} C_DIS
LIN {X 0.164,Y -587.587,Z 1275.164,A 0.000,B 0.000,C 90.000,E1 65.537} C_DIS
LIN {X 0.024,Y -588.809,Z 1275.155,A 0.000,B 0.000,C 90.000,E1 63.948} C_DIS
LIN {X -0.099,Y -590.195,Z 1275.146,A 0.000,B 0.000,C 90.000,E1 62.359} C_DIS
LIN {X 0.065,Y -591.701,Z 1275.138,A 0.000,B 0.000,C 90.000,E1 60.745} C_DIS
LIN {X 0.028,Y -593.367,Z 1275.129,A 0.000,B 0.000,C 90.000,E1 59.154} C_DIS
LIN {X -0.063,Y -594.777,Z 1275.121,A 0.000,B 0.000,C 90.000,E1 57.837} C_DIS
LIN {X 0.178,Y -596.670,Z 1275.111,A 0.000,B 0.000,C 90.000,E1 55.960} C_DIS
LIN {X -0.101,Y -598.219,Z 1275.102,A 0.000,B 0.000,C 90.000,E1 54.402} C_DIS
LIN {X -0.342,Y -599.551,Z 1275.093,A 0.000,B 0.000,C 90.000,E1 52.844} C_DIS
LIN {X 0.044,Y -601.021,Z 1275.083,A 0.000,B 0.000,C 90.000,E1 50.964} C_DIS
LIN {X -0.150,Y -601.555,Z 1275.079,A 0.000,B 0.000,C 90.000,E1 50.194} C_DIS
LIN {X 0.128,Y -601.932,Z 1275.074,A 0.000,B 0.000,C 90.000,E1 49.380} C_DIS
LIN {X -0.219,Y -602.591,Z 1275.066,A 0.000,B 0.000,C 90.000,E1 47.838} C_DIS
LIN {X 0.062,Y -603.058,Z 1275.058,A 0.000,B 0.000,C 90.000,E1 46.500} C_DIS
LIN {X -0.305,Y -603.222,Z 1275.053,A 0.000,B 0.000,C 90.000,E1 45.486} C_DIS
LIN {X -0.251,Y -603.193,Z 1275.047,A 0.000,B 0.000,C 90.000,E1 44.433} C_DIS
LIN {X 0.034,Y -602.942,Z 1275.039,A 0.000,B 0.000,C 90.000,E1 43.095} C_DIS
LIN {X 0.106,Y -602.402,Z 1275.031,A 0.000,B 0.000,C 90.000,E1 41.515} C_DIS
LIN {X 0.175,Y -601.943,Z 1275.025,A 0.000,B 0.000,C 90.000,E1 40.458} C_DIS
LIN {X -0.362,Y -601.322,Z 1275.018,A 0.000,B 0.000,C 90.000,E1 39.197} C_DIS
LIN {X -0.069,Y -600.403,Z 1275.010,A 0.000,B 0.000,C 90.000,E1 37.855} C_DIS
LIN {X 0.065,Y -599.322,Z 1275.005,A 0.000,B 0.000,C 90.000,E1 36.790} C_DIS
LIN {X 0.189,Y -597.996,Z 1274.999,A 0.000,B 0.000,C 90.000,E1 35.724} C_DIS
LIN {X 0.059,Y -596.845,Z 1274.994,A 0.000,B 0.000,C 90.000,E1 34.945} C_DIS
LIN {X -0.197,Y -594.935,Z 1274.988,A 0.000,B 0.000,C 90.000,E1 33.913} C_DIS
LIN {X 0.132,Y -593.450,Z 1274.984,A 0.000,B 0.000,C 90.000,E1 33.086} C_DIS
LIN {X 0.329,Y -590.740,Z 1274.978,A 0.000,B 0.000,C 90.000,E1 32.005} C_DIS
LIN {X -0.204,Y -588.592,Z 1274.974,A 0.000,B 0.000,C 90.000,E1 31.258} C_DIS
LIN {X -0.255,Y -585.978,Z 1274.969,A 0.000,B 0.000,C 90.000,E1 30.463} C_DIS
LIN {X -0.206,Y -584.050,Z 1274.966,A 0.000,B 0.000,C 90.000,E1 29.922} C_DIS
LIN {X 0.202,Y -580.631,Z 1274.962,A 0.000,B 0.000,C 90.000,E1 29.077} C_DIS
LIN {X 0.063,Y -576.991,Z 1274.957,A 0.000,B 0.000,C 90.000,E1 28.281} C_DIS
LIN {X -0.120,Y -570.480,Z 1274.950,A 0.000,B 0.000,C 90.000,E1 27.078} C_DIS
LIN {X 0.041,Y -564.569,Z 1274.945,A 0.000,B 0.000,C 90.000,E1 26.104} C_DIS
LIN {X 0.074,Y -560.023,Z 1274.941,A 0.000,B 0.000,C 90.000,E1 25.412} C_DIS
LIN {X 0.072,Y -555.025,Z 1274.937,A 0.000,B 0.000,C 90.000,E1 24.719} C_DIS
LIN {X 0.138,Y -550.767,Z 1274.934,A 0.000,B 0.000,C 90.000,E1 24.155} C_DIS
LIN {X 0.174,Y -546.191,Z 1274.931,A 0.000,B 0.000,C 90.000,E1 23.590} C_DIS
LIN {X -0.197,Y -540.472,Z 1274.927,A 0.000,B 0.000,C 90.000,E1 22.950} C_DIS
LIN {X 0.166,Y -534.138,Z 1274.923,A 0.000,B 0.000,C 90.000,E1 22.206} C_DIS
LIN {X -0.241,Y -526.278,Z 1274.919,A 0.000,B 0.000,C 90.000,E1 21.408} C_DIS
LIN {X -0.041,Y -515.857,Z 1274.913,A 0.000,B 0.000,C 90.000,E1 20.301} C_DIS
LIN {X -0.114,Y -504.962,Z 1274.907,A 0.000,B 0.000,C 90.000,E1 19.214} C_DIS
LIN {X 0.026,Y -492.500,Z 1274.900,A 0.000,B 0.000,C 90.000,E1 18.000} C_DIS
LIN {X 0.057,Y -486.791,Z 1274.897,A 0.000,B 0.000,C 90.000,E1 17.457} C_DIS
LIN {X -0.047,Y -476.489,Z 1274.892,A 0.000,B 0.000,C 90.000,E1 16.551} C_DIS
LIN {X 0.071,Y -464.666,Z 1274.886,A 0.000,B 0.000,C 90.000,E1 15.481} C_DIS
LIN {X -0.109,Y -446.925,Z 1274.877,A 0.000,B 0.000,C 90.000,E1 13.883} C_DIS
LIN {X 0.011,Y -425.125,Z 1274.865,A 0.000,B 0.000,C 90.000,E1 11.715} C_DIS
LIN {X 0.150,Y -407.949,Z 1274.855,A 0.000,B 0.000,C 90.000,E1 9.849} C_DIS
LIN {X -0.039,Y -399.429,Z 1274.850,A 0.000,B 0.000,C 90.000,E1 8.916} C_DIS
LIN {X 0.071,Y -395.605,Z 1274.846,A 0.000,B 0.000,C 90.000,E1 8.341} C_DIS
LIN {X 0.202,Y -394.958,Z 1274.846,A 0.000,B 0.000,C 90.000,E1 8.163} C_DIS
LIN {X 0.165,Y -394.952,Z 1274.846,A 0.000,B 0.000,C 90.000,E1 8.163} C_DIS
LIN {X 0.110,Y -395.273,Z 1274.845,A 0.000,B 0.000,C 90.000,E1 8.049} C_DIS
LIN {X -0.174,Y -396.256,Z 1274.844,A 0.000,B 0.000,C 90.000,E1 7.936} C_DIS
LIN {X 0.153,Y -399.972,Z 1274.842,A 0.000,B 0.000,C 90.000,E1 7.530} C_DIS
LIN {X -0.164,Y -411.513,Z 1274.838,A 0.000,B 0.000,C 90.000,E1 6.891} C_DIS
LIN {X 0.142,Y -417.874,Z 1274.836,A 0.000,B 0.000,C 90.000,E1 6.429} C_DIS
LIN {X 0.165,Y -425.699,Z 1274.833,A 0.000,B 0.000,C 90.000,E1 5.853} C_DIS
LIN {X -0.151,Y -435.156,Z 1274.829,A 0.000,B 0.000,C 90.000,E1 5.163} C_DIS
LIN {X -0.075,Y -442.943,Z 1274.825,A 0.000,B 0.000,C 90.000,E1 4.531} C_DIS
LIN {X 0.207,Y -452.218,Z 1274.821,A 0.000,B 0.000,C 90.000,E1 3.726} C_DIS
LIN {X 0.013,Y -459.751,Z 1274.817,A 0.000,B 0.000,C 90.000,E1 3.094} C_DIS
LIN {X -0.218,Y -466.695,Z 1274.814,A 0.000,B 0.000,C 90.000,E1 2.465} C_DIS
LIN {X 0.066,Y -473.612,Z 1274.810,A 0.000,B 0.000,C 90.000,E1 1.718} C_DIS
LIN {X 0.159,Y -480.223,Z 1274.806,A 0.000,B 0.000,C 90.000,E1 0.974} C_DIS
LIN {X -0.068,Y -486.661,Z 1274.801,A 0.000,B 0.000,C 90.000,E1 0.229} C_DIS
LIN {X 0.021,Y -492.277,Z 1274.797,A 0.000,B 0.000,C 90.000,E1 359.484} C_DIS
LIN {X -0.105,Y -497.592,Z 1274.793,A 0.000,B 0.000,C 90.000,E1 358.740} C_DIS
LIN {X 0.021,Y -503.437,Z 1274.788,A 0.000,B 0.000,C 90.000,E1 357.822} C_DIS
LIN {X -0.008,Y -507.969,Z 1274.784,A 0.000,B 0.000,C 90.000,E1 357.078} C_DIS
LIN {X -0.180,Y -511.418,Z 1274.781,A 0.000,B 0.000,C 90.000,E1 356.502} C_DIS
LIN {X -0.108,Y -515.432,Z 1274.776,A 0.000,B 0.000,C 90.000,E1 355.755} C_DIS
LIN {X -0.220,Y -518.432,Z 1274.773,A 0.000,B 0.000,C 90.000,E1 355.179} C_DIS
LIN {X 0.148,Y -522.636,Z 1274.768,A 0.000,B 0.000,C 90.000,E1 354.261} C_DIS
LIN {X 0.094,Y -526.529,Z 1274.763,A 0.000,B 0.000,C 90.000,E1 353.394} C_DIS
LIN {X -0.203,Y -530.513,Z 1274.758,A 0.000,B 0.000,C 90.000,E1 352.413} C_DIS
LIN {X -0.176,Y -533.681,Z 1274.753,A 0.000,B 0.000,C 90.000,E1 351.546} C_DIS
LIN {X -0.119,Y -536.537,Z 1274.748,A 0.000,B 0.000,C 90.000,E1 350.679} C_DIS
LIN {X 0.059,Y -539.090,Z 1274.743,A 0.000,B 0.000,C 90.000,E1 349.803} C_DIS
LIN {X -0.291,Y -542.240,Z 1274.737,A 0.000,B 0.000,C 90.000,E1 348.701} C_DIS
LIN {X 0.152,Y -544.908,Z 1274.731,A 0.000,B 0.000,C 90.000,E1 347.521} C_DIS
LIN {X -0.107,Y -546.756,Z 1274.726,A 0.000,B 0.000,C 90.000,E1 346.700} C_DIS
LIN {X 0.180,Y -548.390,Z 1274.721,A 0.000,B 0.000,C 90.000,E1 345.825} C_DIS
LIN {X 0.187,Y -550.278,Z 1274.715,A 0.000,B 0.000,C 90.000,E1 344.700} C_DIS
LIN {X -0.158,Y -551.833,Z 1274.709,A 0.000,B 0.000,C 90.000,E1 343.614} C_DIS
LIN {X -0.108,Y -553.060,Z 1274.703,A 0.000,B 0.000,C 90.000,E1 342.489} C_DIS
LIN {X 0.117,Y -553.834,Z 1274.697,A 0.000,B 0.000,C 90.000,E1 341.348} C_DIS
LIN {X -0.273,Y -554.116,Z 1274.692,A 0.000,B 0.000,C 90.000,E1 340.550} C_DIS
LIN {X 0.294,Y -554.082,Z 1274.689,A 0.000,B 0.000,C 90.000,E1 339.934} C_DIS
LIN {X -0.084,Y -553.760,Z 1274.684,A 0.000,B 0.000,C 90.000,E1 339.135} C_DIS
LIN {X -0.181,Y -552.899,Z 1274.678,A 0.000,B 0.000,C 90.000,E1 338.028} C_DIS
LIN {X -0.341,Y -552.220,Z 1274.675,A 0.000,B 0.000,C 90.000,E1 337.486} C_DIS
LIN {X -0.022,Y -550.996,Z 1274.670,A 0.000,B 0.000,C 90.000,E1 336.613} C_DIS
LIN {X -0.193,Y -548.427,Z 1274.662,A 0.000,B 0.000,C 90.000,E1 335.229} C_DIS
LIN {X 0.067,Y -547.857,Z 1274.661,A 0.000,B 0.000,C 90.000,E1 334.921} C_DIS
LIN {X 0.072,Y -545.708,Z 1274.656,A 0.000,B 0.000,C 90.000,E1 334.076} C_DIS
LIN {X -0.180,Y -543.348,Z 1274.651,A 0.000,B 0.000,C 90.000,E1 333.256} C_DIS
LIN {X -0.212,Y -540.608,Z 1274.647,A 0.000,B 0.000,C 90.000,E1 332.410} C_DIS
LIN {X 0.202,Y -537.338,Z 1274.642,A 0.000,B 0.000,C 90.000,E1 331.513} C_DIS
LIN {X 0.102,Y -533.592,Z 1274.637,A 0.000,B 0.000,C 90.000,E1 330.667} C_DIS
LIN {X 0.101,Y -530.062,Z 1274.633,A 0.000,B 0.000,C 90.000,E1 329.950} C_DIS
LIN {X 0.176,Y -525.104,Z 1274.628,A 0.000,B 0.000,C 90.000,E1 329.076} C_DIS
LIN {X -0.027,Y -517.386,Z 1274.621,A 0.000,B 0.000,C 90.000,E1 327.788} C_DIS
LIN {X -0.087,Y -512.182,Z 1274.616,A 0.000,B 0.000,C 90.000,E1 326.914} C_DIS
LIN {X -0.118,Y -507.308,Z 1274.611,A 0.000,B 0.000,C 90.000,E1 325.928} C_DIS
LIN {X 0.011,Y -505.373,Z 1274.608,A 0.000,B 0.000,C 90.000,E1 325.468} C_DIS
LIN {X -0.093,Y -504.288,Z 1274.607,A 0.000,B 0.000,C 90.000,E1 325.182} C_DIS
LIN {X -0.009,Y -501.903,Z 1274.602,A 0.000,B 0.000,C 90.000,E1 324.276} C_DIS
LIN {X 0.043,Y -500.294,Z 1274.597,A 0.000,B 0.000,C 90.000,E1 323.371} C_DIS
LIN {X -0.146,Y -499.305,Z 1274.590,A 0.000,B 0.000,C 90.000,E1 322.190} C_DIS
LIN {X 0.105,Y -498.906,Z 1274.580,A 0.000,B 0.000,C 90.000,E1 320.356} C_DIS
LIN {X 0.157,Y -499.195,Z 1274.568,A 0.000,B 0.000,C 90.000,E1 318.243} C_DIS
LIN {X 0.115,Y -499.470,Z 1274.560,A 0.000,B 0.000,C 90.000,E1 316.743} C_DIS
LIN {X 0.080,Y -499.688,Z 1274.551,A 0.000,B 0.000,C 90.000,E1 315.243} C_DIS
LIN {X 0.049,Y -500.003,Z 1274.543,A 0.000,B 0.000,C 90.000,E1 313.743} C_DIS
LIN {X -0.274,Y -500.441,Z 1274.531,A 0.000,B 0.000,C 90.000,E1 311.676} C_DIS
LIN {X -0.002,Y -500.635,Z 1274.526,A 0.000,B 0.000,C 90.000,E1 310.744} C_DIS
LIN {X 0.035,Y -500.913,Z 1274.513,A 0.000,B 0.000,C 90.000,E1 308.338} C_DIS
LIN {X -0.256,Y -501.119,Z 1274.505,A 0.000,B 0.000,C 90.000,E1 306.870} C_DIS
LIN {X 0.253,Y -501.313,Z 1274.496,A 0.000,B 0.000,C 90.000,E1 305.311} C_DIS
LIN {X 0.061,Y -501.341,Z 1274.488,A 0.000,B 0.000,C 90.000,E1 303.833} C_DIS
LIN {X -0.167,Y -501.128,Z 1274.483,A 0.000,B 0.000,C 90.000,E1 302.959} C_DIS
LIN {X -0.095,Y -500.500,Z 1274.476,A 0.000,B 0.000,C 90.000,E1 301.750} C_DIS
LIN {X 0.069,Y -499.981,Z 1274.473,A 0.000,B 0.000,C 90.000,E1 301.131} C_DIS
LIN {X -0.030,Y -499.269,Z 1274.470,A 0.000,B 0.000,C 90.000,E1 300.541} C_DIS
LIN {X 0.118,Y -498.297,Z 1274.466,A 0.000,B 0.000,C 90.000,E1 299.922} C_DIS
LIN {X 0.156,Y -497.670,Z 1274.465,A 0.000,B 0.000,C 90.000,E1 299.617} C_DIS
LIN {X 0.007,Y -496.863,Z 1274.463,A 0.000,B 0.000,C 90.000,E1 299.333} C_DIS
LIN {X 0.046,Y -495.676,Z 1274.461,A 0.000,B 0.000,C 90.000,E1 299.027} C_DIS
LIN {X 0.061,Y -481.926,Z 1274.444,A 0.000,B 0.000,C 90.000,E1 295.976} C_DIS
LIN {X -0.167,Y -470.031,Z 1274.427,A 0.000,B 0.000,C 90.000,E1 292.898} C_DIS
LIN {X 0.051,Y -458.978,Z 1274.408,A 0.000,B 0.000,C 90.000,E1 289.396} C_DIS
LIN {X 0.230,Y -449.954,Z 1274.388,A 0.000,B 0.000,C 90.000,E1 285.843} C_DIS
LIN {X -0.115,Y -441.800,Z 1274.365,A 0.000,B 0.000,C 90.000,E1 281.658} C_DIS
LIN {X 0.034,Y -435.361,Z 1274.335,A 0.000,B 0.000,C 90.000,E1 276.372} C_DIS
LIN {X 0.072,Y -436.401,Z 1274.260,A 0.000,B 0.000,C 90.000,E1 262.761} C_DIS
LIN {X 0.053,Y -443.115,Z 1274.232,A 0.000,B 0.000,C 90.000,E1 257.825} C_DIS
LIN {X 0.028,Y -451.025,Z 1274.211,A 0.000,B 0.000,C 90.000,E1 253.921} C_DIS
LIN {X 0.150,Y -460.340,Z 1274.191,A 0.000,B 0.000,C 90.000,E1 250.369} C_DIS
LIN {X 0.070,Y -467.333,Z 1274.179,A 0.000,B 0.000,C 90.000,E1 248.156} C_DIS
LIN {X 0.011,Y -468.184,Z 1274.177,A 0.000,B 0.000,C 90.000,E1 247.847} C_DIS
LIN {X -0.043,Y -468.697,Z 1274.175,A 0.000,B 0.000,C 90.000,E1 247.539} C_DIS
LIN {X -0.144,Y -469.330,Z 1274.172,A 0.000,B 0.000,C 90.000,E1 246.922} C_DIS
LIN {X -0.054,Y -469.640,Z 1274.168,A 0.000,B 0.000,C 90.000,E1 246.282} C_DIS
LIN {X -0.196,Y -469.754,Z 1274.163,A 0.000,B 0.000,C 90.000,E1 245.357} C_DIS
LIN {X 0.005,Y -469.413,Z 1274.156,A 0.000,B 0.000,C 90.000,E1 244.076} C_DIS
LIN {X -0.008,Y -468.730,Z 1274.149,A 0.000,B 0.000,C 90.000,E1 242.820} C_DIS
LIN {X -0.264,Y -467.366,Z 1274.135,A 0.000,B 0.000,C 90.000,E1 240.333} C_DIS
LIN {X -0.139,Y -466.413,Z 1274.126,A 0.000,B 0.000,C 90.000,E1 238.742} C_DIS
LIN {X -0.086,Y -465.803,Z 1274.121,A 0.000,B 0.000,C 90.000,E1 237.788} C_DIS
LIN {X -0.001,Y -464.499,Z 1274.110,A 0.000,B 0.000,C 90.000,E1 235.881} C_DIS
LIN {X -0.167,Y -462.841,Z 1274.095,A 0.000,B 0.000,C 90.000,E1 233.050} C_DIS
LIN {X 0.027,Y -461.816,Z 1274.082,A 0.000,B 0.000,C 90.000,E1 230.803} C_DIS
LIN {X 0.160,Y -460.891,Z 1274.068,A 0.000,B 0.000,C 90.000,E1 228.243} C_DIS
LIN {X -0.157,Y -460.232,Z 1274.056,A 0.000,B 0.000,C 90.000,E1 226.053} C_DIS
LIN {X 0.148,Y -459.712,Z 1274.043,A 0.000,B 0.000,C 90.000,E1 223.785} C_DIS
LIN {X 0.075,Y -459.900,Z 1274.022,A 0.000,B 0.000,C 90.000,E1 219.967} C_DIS
LIN {X -0.005,Y -461.651,Z 1273.997,A 0.000,B 0.000,C 90.000,E1 215.518} C_DIS
LIN {X 0.023,Y -464.506,Z 1273.980,A 0.000,B 0.000,C 90.000,E1 212.339} C_DIS
LIN {X -0.149,Y -466.746,Z 1273.969,A 0.000,B 0.000,C 90.000,E1 210.463} C_DIS
LIN {X -0.096,Y -468.985,Z 1273.959,A 0.000,B 0.000,C 90.000,E1 208.565} C_DIS
LIN {X 0.066,Y -472.454,Z 1273.943,A 0.000,B 0.000,C 90.000,E1 205.720} C_DIS
LIN {X 0.165,Y -476.578,Z 1273.927,A 0.000,B 0.000,C 90.000,E1 202.898} C_DIS
LIN {X 0.057,Y -480.081,Z 1273.915,A 0.000,B 0.000,C 90.000,E1 200.737} C_DIS
LIN {X -0.137,Y -484.442,Z 1273.902,A 0.000,B 0.000,C 90.000,E1 198.290} C_DIS
LIN {X -0.073,Y -488.427,Z 1273.890,A 0.000,B 0.000,C 90.000,E1 196.134} C_DIS
LIN {X -0.053,Y -491.845,Z 1273.880,A 0.000,B 0.000,C 90.000,E1 194.300} C_DIS
LIN {X -0.051,Y -496.035,Z 1273.868,A 0.000,B 0.000,C 90.000,E1 192.175} C_DIS
LIN {X 0.004,Y -499.023,Z 1273.859,A 0.000,B 0.000,C 90.000,E1 190.658} C_DIS
LIN {X -0.039,Y -502.580,Z 1273.849,A 0.000,B 0.000,C 90.000,E1 188.859} C_DIS
LIN {X -0.069,Y -506.302,Z 1273.839,A 0.000,B 0.000,C 90.000,E1 187.068} C_DIS
LIN {X 0.036,Y -509.243,Z 1273.831,A 0.000,B 0.000,C 90.000,E1 185.568} C_DIS
LIN {X 0.008,Y -513.347,Z 1273.819,A 0.000,B 0.000,C 90.000,E1 183.498} C_DIS
LIN {X 0.164,Y -516.168,Z 1273.811,A 0.000,B 0.000,C 90.000,E1 182.007} C_DIS
LIN {X -0.148,Y -518.876,Z 1273.803,A 0.000,B 0.000,C 90.000,E1 180.573} C_DIS
LIN {X 0.048,Y -521.951,Z 1273.793,A 0.000,B 0.000,C 90.000,E1 178.797} C_DIS
LIN {X -0.122,Y -523.850,Z 1273.787,A 0.000,B 0.000,C 90.000,E1 177.650} C_DIS
LIN {X 0.266,Y -525.641,Z 1273.781,A 0.000,B 0.000,C 90.000,E1 176.445} C_DIS
LIN {X 0.148,Y -527.236,Z 1273.774,A 0.000,B 0.000,C 90.000,E1 175.298} C_DIS
LIN {X 0.094,Y -528.615,Z 1273.768,A 0.000,B 0.000,C 90.000,E1 174.147} C_DIS
LIN {X 0.058,Y -529.832,Z 1273.761,A 0.000,B 0.000,C 90.000,E1 172.996} C_DIS
LIN {X 0.138,Y -531.002,Z 1273.753,A 0.000,B 0.000,C 90.000,E1 171.546} C_DIS
LIN {X 0.207,Y -531.710,Z 1273.747,A 0.000,B 0.000,C 90.000,E1 170.387} C_DIS
LIN {X -0.147,Y -532.173,Z 1273.740,A 0.000,B 0.000,C 90.000,E1 169.275} C_DIS
LIN {X -0.075,Y -532.452,Z 1273.734,A 0.000,B 0.000,C 90.000,E1 168.117} C_DIS
LIN {X 0.171,Y -532.521,Z 1273.729,A 0.000,B 0.000,C 90.000,E1 167.229} C_DIS
LIN {X -0.173,Y -532.478,Z 1273.723,A 0.000,B 0.000,C 90.000,E1 166.117} C_DIS
LIN {X 0.040,Y -532.314,Z 1273.710,A 0.000,B 0.000,C 90.000,E1 163.795} C_DIS
LIN {X 0.189,Y -532.446,Z 1273.700,A 0.000,B 0.000,C 90.000,E1 162.054} C_DIS
LIN {X 0.031,Y -533.721,Z 1273.689,A 0.000,B 0.000,C 90.000,E1 160.061} C_DIS
LIN {X -0.050,Y -534.938,Z 1273.685,A 0.000,B 0.000,C 90.000,E1 159.209} C_DIS
LIN {X 0.087,Y -537.229,Z 1273.678,A 0.000,B 0.000,C 90.000,E1 158.050} C_DIS
LIN {X 0.017,Y -538.784,Z 1273.675,A 0.000,B 0.000,C 90.000,E1 157.486} C_DIS
LIN {X -0.080,Y -542.681,Z 1273.669,A 0.000,B 0.000,C 90.000,E1 156.357} C_DIS
LIN {X -0.232,Y -546.043,Z 1273.665,A 0.000,B 0.000,C 90.000,E1 155.665} C_DIS
LIN {X 0.144,Y -549.850,Z 1273.661,A 0.000,B 0.000,C 90.000,E1 154.921} C_DIS
LIN {X 0.055,Y -554.111,Z 1273.657,A 0.000,B 0.000,C 90.000,E1 154.229} C_DIS
LIN {X -0.064,Y -561.872,Z 1273.651,A 0.000,B 0.000,C 90.000,E1 153.127} C_DIS
LIN {X 0.208,Y -567.382,Z 1273.647,A 0.000,B 0.000,C 90.000,E1 152.410} C_DIS
LIN {X -0.322,Y -574.256,Z 1273.642,A 0.000,B 0.000,C 90.000,E1 151.641} C_DIS
LIN {X 0.024,Y -581.989,Z 1273.637,A 0.000,B 0.000,C 90.000,E1 150.667} C_DIS
LIN {X 0.009,Y -590.783,Z 1273.631,A 0.000,B 0.000,C 90.000,E1 149.616} C_DIS
LIN {X 0.090,Y -595.055,Z 1273.628,A 0.000,B 0.000,C 90.000,E1 149.076} C_DIS
LIN {X -0.207,Y -601.935,Z 1273.623,A 0.000,B 0.000,C 90.000,E1 148.201} C_DIS
LIN {X 0.296,Y -607.617,Z 1273.619,A 0.000,B 0.000,C 90.000,E1 147.375} C_DIS
LIN {X -0.067,Y -612.901,Z 1273.615,A 0.000,B 0.000,C 90.000,E1 146.628} C_DIS
LIN {X 0.187,Y -617.106,Z 1273.611,A 0.000,B 0.000,C 90.000,E1 145.960} C_DIS
LIN {X -0.058,Y -620.210,Z 1273.608,A 0.000,B 0.000,C 90.000,E1 145.468} C_DIS
LIN {X 0.060,Y -623.826,Z 1273.605,A 0.000,B 0.000,C 90.000,E1 144.815} C_DIS
LIN {X -0.138,Y -626.616,Z 1273.602,A 0.000,B 0.000,C 90.000,E1 144.322} C_DIS
LIN {X 0.031,Y -631.157,Z 1273.597,A 0.000,B 0.000,C 90.000,E1 143.417} C_DIS
LIN {X 0.111,Y -636.256,Z 1273.590,A 0.000,B 0.000,C 90.000,E1 142.271} C_DIS
LIN {X 0.159,Y -641.248,Z 1273.583,A 0.000,B 0.000,C 90.000,E1 141.009} C_DIS
LIN {X -0.118,Y -644.808,Z 1273.578,A 0.000,B 0.000,C 90.000,E1 140.033} C_DIS
LIN {X 0.074,Y -648.879,Z 1273.571,A 0.000,B 0.000,C 90.000,E1 138.771} C_DIS
LIN {X -0.168,Y -652.832,Z 1273.564,A 0.000,B 0.000,C 90.000,E1 137.553} C_DIS
LIN {X 0.132,Y -655.744,Z 1273.559,A 0.000,B 0.000,C 90.000,E1 136.539} C_DIS
LIN {X -0.076,Y -660.906,Z 1273.549,A 0.000,B 0.000,C 90.000,E1 134.838} C_DIS
LIN {X -0.164,Y -665.532,Z 1273.541,A 0.000,B 0.000,C 90.000,E1 133.380} C_DIS
LIN {X -0.134,Y -670.108,Z 1273.533,A 0.000,B 0.000,C 90.000,E1 131.919} C_DIS
LIN {X -0.028,Y -673.824,Z 1273.526,A 0.000,B 0.000,C 90.000,E1 130.701} C_DIS
LIN {X 0.136,Y -677.389,Z 1273.519,A 0.000,B 0.000,C 90.000,E1 129.483} C_DIS
LIN {X -0.082,Y -680.821,Z 1273.513,A 0.000,B 0.000,C 90.000,E1 128.302} C_DIS
LIN {X -0.280,Y -683.439,Z 1273.507,A 0.000,B 0.000,C 90.000,E1 127.363} C_DIS
LIN {X 0.105,Y -685.944,Z 1273.502,A 0.000,B 0.000,C 90.000,E1 126.377} C_DIS
LIN {X 0.190,Y -689.390,Z 1273.494,A 0.000,B 0.000,C 90.000,E1 124.945} C_DIS
LIN {X 0.265,Y -691.549,Z 1273.489,A 0.000,B 0.000,C 90.000,E1 123.992} C_DIS
LIN {X 0.020,Y -693.921,Z 1273.482,A 0.000,B 0.000,C 90.000,E1 122.832} C_DIS
LIN {X -0.188,Y -696.156,Z 1273.476,A 0.000,B 0.000,C 90.000,E1 121.671} C_DIS
LIN {X 0.227,Y -698.188,Z 1273.469,A 0.000,B 0.000,C 90.000,E1 120.463} C_DIS
LIN {X -0.287,Y -699.954,Z 1273.463,A 0.000,B 0.000,C 90.000,E1 119.333} C_DIS
LIN {X -0.096,Y -700.901,Z 1273.459,A 0.000,B 0.000,C 90.000,E1 118.615} C_DIS
LIN {X 0.380,Y -701.970,Z 1273.454,A 0.000,B 0.000,C 90.000,E1 117.641} C_DIS
LIN {X -0.356,Y -702.537,Z 1273.450,A 0.000,B 0.000,C 90.000,E1 117.001} C_DIS
LIN {X -0.145,Y -702.756,Z 1273.446,A 0.000,B 0.000,C 90.000,E1 116.283} C_DIS
LIN {X 0.108,Y -702.792,Z 1273.443,A 0.000,B 0.000,C 90.000,E1 115.796} C_DIS
LIN {X 0.315,Y -702.438,Z 1273.440,A 0.000,B 0.000,C 90.000,E1 115.079} C_DIS
LIN {X -0.062,Y -702.034,Z 1273.437,A 0.000,B 0.000,C 90.000,E1 114.643} C_DIS
LIN {X 0.203,Y -701.317,Z 1273.434,A 0.000,B 0.000,C 90.000,E1 114.155} C_DIS
LIN {X -0.163,Y -700.617,Z 1273.433,A 0.000,B 0.000,C 90.000,E1 113.951} C_DIS
LIN {X 0.097,Y -698.755,Z 1273.430,A 0.000,B 0.000,C 90.000,E1 113.462} C_DIS
LIN {X 0.231,Y -698.004,Z 1273.430,A 0.000,B 0.000,C 90.000,E1 113.334} C_DIS
LIN {X -0.293,Y -695.069,Z 1273.428,A 0.000,B 0.000,C 90.000,E1 113.025} C_DIS
LIN {X -0.267,Y -693.272,Z 1273.427,A 0.000,B 0.000,C 90.000,E1 112.823} C_DIS
LIN {X -0.144,Y -691.483,Z 1273.426,A 0.000,B 0.000,C 90.000,E1 112.695} C_DIS
LIN {X -0.287,Y -688.877,Z 1273.425,A 0.000,B 0.000,C 90.000,E1 112.589} C_DIS
LIN {X -0.044,Y -682.660,Z 1273.424,A 0.000,B 0.000,C 90.000,E1 112.333} C_DIS
LIN {X -0.220,Y -680.379,Z 1273.424,A 0.000,B 0.000,C 90.000,E1 112.280} C_DIS
LIN {X -0.137,Y -676.891,Z 1273.423,A 0.000,B 0.000,C 90.000,E1 112.206} C_DIS
LIN {X -0.281,Y -669.872,Z 1273.423,A 0.000,B 0.000,C 90.000,E1 112.153} C_DIS
LIN {X -0.316,Y -636.704,Z 1273.423,A 0.000,B 0.000,C 90.000,E1 112.153} C_DIS
LIN {X -0.085,Y -633.707,Z 1273.422,A 0.000,B 0.000,C 90.000,E1 112.025} C_DIS
LIN {X -0.128,Y -633.634,Z 1273.422,A 0.000,B 0.000,C 90.000,E1 112.025} C_DIS
LIN {X 0.323,Y -634.391,Z 1273.421,A 0.000,B 0.000,C 90.000,E1 111.716} C_DIS
LIN {X 0.257,Y -635.746,Z 1273.419,A 0.000,B 0.000,C 90.000,E1 111.461} C_DIS
LIN {X 0.091,Y -644.090,Z 1273.413,A 0.000,B 0.000,C 90.000,E1 110.301} C_DIS
LIN {X 0.013,Y -648.087,Z 1273.409,A 0.000,B 0.000,C 90.000,E1 109.685} C_DIS
LIN {X -0.177,Y -652.771,Z 1273.405,A 0.000,B 0.000,C 90.000,E1 108.833} C_DIS
LIN {X 0.222,Y -655.860,Z 1273.401,A 0.000,B 0.000,C 90.000,E1 108.181} C_DIS
LIN {X 0.070,Y -659.224,Z 1273.397,A 0.000,B 0.000,C 90.000,E1 107.457} C_DIS
LIN {X -0.055,Y -662.318,Z 1273.393,A 0.000,B 0.000,C 90.000,E1 106.732} C_DIS
LIN {X -0.250,Y -664.250,Z 1273.390,A 0.000,B 0.000,C 90.000,E1 106.260} C_DIS
LIN {X 0.212,Y -665.967,Z 1273.388,A 0.000,B 0.000,C 90.000,E1 105.733} C_DIS
LIN {X 0.146,Y -668.118,Z 1273.384,A 0.000,B 0.000,C 90.000,E1 105.009} C_DIS
LIN {X -0.005,Y -669.316,Z 1273.381,A 0.000,B 0.000,C 90.000,E1 104.537} C_DIS
LIN {X -0.217,Y -670.661,Z 1273.377,A 0.000,B 0.000,C 90.000,E1 103.828} C_DIS
LIN {X 0.302,Y -671.364,Z 1273.374,A 0.000,B 0.000,C 90.000,E1 103.300} C_DIS
LIN {X 0.109,Y -671.898,Z 1273.370,A 0.000,B 0.000,C 90.000,E1 102.591} C_DIS
LIN {X -0.019,Y -672.130,Z 1273.367,A 0.000,B 0.000,C 90.000,E1 102.119} C_DIS
LIN {X -0.348,Y -671.891,Z 1273.363,A 0.000,B 0.000,C 90.000,E1 101.422} C_DIS
LIN {X 0.181,Y -671.578,Z 1273.361,A 0.000,B 0.000,C 90.000,E1 100.894} C_DIS
LIN {X -0.077,Y -671.018,Z 1273.358,A 0.000,B 0.000,C 90.000,E1 100.433} C_DIS
LIN {X -0.218,Y -670.170,Z 1273.355,A 0.000,B 0.000,C 90.000,E1 99.962} C_DIS
LIN {X 0.181,Y -669.114,Z 1273.353,A 0.000,B 0.000,C 90.000,E1 99.443} C_DIS
LIN {X 0.022,Y -667.722,Z 1273.350,A 0.000,B 0.000,C 90.000,E1 98.973} C_DIS
LIN {X -0.165,Y -666.933,Z 1273.349,A 0.000,B 0.000,C 90.000,E1 98.746} C_DIS
LIN {X 0.316,Y -665.040,Z 1273.346,A 0.000,B 0.000,C 90.000,E1 98.219} C_DIS
LIN {X -0.070,Y -662.217,Z 1273.343,A 0.000,B 0.000,C 90.000,E1 97.644} C_DIS
LIN {X 0.183,Y -658.828,Z 1273.339,A 0.000,B 0.000,C 90.000,E1 97.011} C_DIS
LIN {X -0.141,Y -655.804,Z 1273.336,A 0.000,B 0.000,C 90.000,E1 96.549} C_DIS
LIN {X 0.166,Y -652.481,Z 1273.334,A 0.000,B 0.000,C 90.000,E1 96.030} C_DIS
LIN {X -0.248,Y -647.647,Z 1273.330,A 0.000,B 0.000,C 90.000,E1 95.448} C_DIS
LIN {X -0.059,Y -643.459,Z 1273.327,A 0.000,B 0.000,C 90.000,E1 94.935} C_DIS
LIN {X 0.157,Y -638.898,Z 1273.325,A 0.000,B 0.000,C 90.000,E1 94.416} C_DIS
LIN {X -0.287,Y -632.658,Z 1273.321,A 0.000,B 0.000,C 90.000,E1 93.841} C_DIS
LIN {X 0.240,Y -627.719,Z 1273.319,A 0.000,B 0.000,C 90.000,E1 93.326} C_DIS
LIN {X 0.166,Y -620.798,Z 1273.315,A 0.000,B 0.000,C 90.000,E1 92.751} C_DIS
LIN {X 0.287,Y -615.126,Z 1273.313,A 0.000,B 0.000,C 90.000,E1 92.293} C_DIS
LIN {X 0.046,Y -607.771,Z 1273.310,A 0.000,B 0.000,C 90.000,E1 91.776} C_DIS
LIN {X -0.203,Y -603.373,Z 1273.308,A 0.000,B 0.000,C 90.000,E1 91.489} C_DIS
LIN {X 0.078,Y -595.431,Z 1273.306,A 0.000,B 0.000,C 90.000,E1 90.974} C_DIS
LIN {X 0.204,Y -590.305,Z 1273.304,A 0.000,B 0.000,C 90.000,E1 90.688} C_DIS
LIN {X -0.098,Y -583.216,Z 1273.302,A 0.000,B 0.000,C 90.000,E1 90.401} C_DIS
LIN {X 0.027,Y -576.234,Z 1273.301,A 0.000,B 0.000,C 90.000,E1 90.115} C_DIS
LIN {X -0.097,Y -572.350,Z 1273.300,A 0.000,B 0.000,C 90.000,E1 89.943} C_DIS
LIN {X 0.030,Y -569.233,Z 1273.298,A 0.000,B 0.000,C 90.000,E1 89.599} C_DIS
LIN {X -0.012,Y -569.220,Z 1273.298,A 0.000,B 0.000,C 90.000,E1 89.599} C_DIS
LIN {X -0.059,Y -568.726,Z 1273.297,A 0.000,B 0.000,C 90.000,E1 89.427} C_DIS
LIN {X -0.069,Y -568.706,Z 1273.293,A 0.000,B 0.000,C 90.000,E1 88.740} C_DIS
LIN {X -0.159,Y -570.385,Z 1273.281,A 0.000,B 0.000,C 90.000,E1 86.560} C_DIS
LIN {X -0.031,Y -572.817,Z 1273.267,A 0.000,B 0.000,C 90.000,E1 84.090} C_DIS
LIN {X -0.163,Y -574.603,Z 1273.258,A 0.000,B 0.000,C 90.000,E1 82.470} C_DIS
LIN {X 0.114,Y -576.181,Z 1273.251,A 0.000,B 0.000,C 90.000,E1 81.084} C_DIS
LIN {X -0.067,Y -577.607,Z 1273.243,A 0.000,B 0.000,C 90.000,E1 79.746} C_DIS
LIN {X 0.234,Y -578.577,Z 1273.237,A 0.000,B 0.000,C 90.000,E1 78.634} C_DIS
LIN {X -0.259,Y -579.943,Z 1273.228,A 0.000,B 0.000,C 90.000,E1 77.061} C_DIS
LIN {X 0.204,Y -580.788,Z 1273.222,A 0.000,B 0.000,C 90.000,E1 75.936} C_DIS
LIN {X -0.212,Y -581.749,Z 1273.215,A 0.000,B 0.000,C 90.000,E1 74.629} C_DIS
LIN {X -0.058,Y -582.528,Z 1273.207,A 0.000,B 0.000,C 90.000,E1 73.268} C_DIS
LIN {X 0.114,Y -583.562,Z 1273.198,A 0.000,B 0.000,C 90.000,E1 71.638} C_DIS
LIN {X 0.241,Y -584.177,Z 1273.192,A 0.000,B 0.000,C 90.000,E1 70.550} C_DIS
LIN {X 0.098,Y -585.022,Z 1273.183,A 0.000,B 0.000,C 90.000,E1 68.954} C_DIS
LIN {X -0.152,Y -586.211,Z 1273.173,A 0.000,B 0.000,C 90.000,E1 67.102} C_DIS
LIN {X -0.035,Y -587.510,Z 1273.164,A 0.000,B 0.000,C 90.000,E1 65.485} C_DIS
LIN {X -0.184,Y -588.755,Z 1273.155,A 0.000,B 0.000,C 90.000,E1 63.896} C_DIS
LIN {X -0.041,Y -590.147,Z 1273.146,A 0.000,B 0.000,C 90.000,E1 62.281} C_DIS
LIN {X 0.128,Y -591.662,Z 1273.137,A 0.000,B 0.000,C 90.000,E1 60.667} C_DIS
LIN {X 0.098,Y -593.336,Z 1273.128,A 0.000,B 0.000,C 90.000,E1 59.076} C_DIS
LIN {X -0.091,Y -595.005,Z 1273.120,A 0.000,B 0.000,C 90.000,E1 57.502} C_DIS
LIN {X 0.256,Y -596.628,Z 1273.111,A 0.000,B 0.000,C 90.000,E1 55.881} C_DIS
LIN {X 0.234,Y -597.929,Z 1273.103,A 0.000,B 0.000,C 90.000,E1 54.562} C_DIS
LIN {X -0.021,Y -599.270,Z 1273.094,A 0.000,B 0.000,C 90.000,E1 53.004} C_DIS
LIN {X 0.111,Y -600.502,Z 1273.086,A 0.000,B 0.000,C 90.000,E1 51.412} C_DIS
LIN {X 0.153,Y -601.333,Z 1273.080,A 0.000,B 0.000,C 90.000,E1 50.356} C_DIS
LIN {X -0.031,Y -601.749,Z 1273.076,A 0.000,B 0.000,C 90.000,E1 49.585} C_DIS
LIN {X -0.134,Y -602.455,Z 1273.065,A 0.000,B 0.000,C 90.000,E1 47.757} C_DIS
LIN {X 0.139,Y -602.778,Z 1273.061,A 0.000,B 0.000,C 90.000,E1 46.944} C_DIS
LIN {X 0.180,Y -603.047,Z 1273.055,A 0.000,B 0.000,C 90.000,E1 45.891} C_DIS
LIN {X 0.230,Y -603.090,Z 1273.049,A 0.000,B 0.000,C 90.000,E1 44.838} C_DIS
LIN {X 0.280,Y -602.976,Z 1273.043,A 0.000,B 0.000,C 90.000,E1 43.785} C_DIS
LIN {X -0.090,Y -602.690,Z 1273.038,A 0.000,B 0.000,C 90.000,E1 42.771} C_DIS
LIN {X 0.179,Y -602.233,Z 1273.030,A 0.000,B 0.000,C 90.000,E1 41.434} C_DIS
LIN {X -0.357,Y -601.646,Z 1273.023,A 0.000,B 0.000,C 90.000,E1 40.172} C_DIS
LIN {X -0.296,Y -601.104,Z 1273.017,A 0.000,B 0.000,C 90.000,E1 39.116} C_DIS
LIN {X -0.379,Y -600.188,Z 1273.010,A 0.000,B 0.000,C 90.000,E1 37.810} C_DIS
LIN {X 0.119,Y -599.086,Z 1273.004,A 0.000,B 0.000,C 90.000,E1 36.710} C_DIS
LIN {X -0.112,Y -597.740,Z 1272.998,A 0.000,B 0.000,C 90.000,E1 35.678} C_DIS
LIN {X -0.239,Y -596.556,Z 1272.994,A 0.000,B 0.000,C 90.000,E1 34.898} C_DIS
LIN {X -0.160,Y -594.648,Z 1272.988,A 0.000,B 0.000,C 90.000,E1 33.833} C_DIS
LIN {X -0.160,Y -593.077,Z 1272.984,A 0.000,B 0.000,C 90.000,E1 33.038} C_DIS
LIN {X 0.149,Y -591.077,Z 1272.979,A 0.000,B 0.000,C 90.000,E1 32.212} C_DIS
LIN {X 0.315,Y -588.168,Z 1272.973,A 0.000,B 0.000,C 90.000,E1 31.131} C_DIS
LIN {X 0.259,Y -585.479,Z 1272.969,A 0.000,B 0.000,C 90.000,E1 30.335} C_DIS
LIN {X 0.304,Y -583.503,Z 1272.966,A 0.000,B 0.000,C 90.000,E1 29.795} C_DIS
LIN {X -0.085,Y -580.061,Z 1272.961,A 0.000,B 0.000,C 90.000,E1 29.027} C_DIS
LIN {X -0.222,Y -576.384,Z 1272.957,A 0.000,B 0.000,C 90.000,E1 28.231} C_DIS
LIN {X -0.066,Y -570.512,Z 1272.951,A 0.000,B 0.000,C 90.000,E1 27.129} C_DIS
LIN {X -0.069,Y -565.539,Z 1272.946,A 0.000,B 0.000,C 90.000,E1 26.309} C_DIS
LIN {X 0.122,Y -560.145,Z 1272.942,A 0.000,B 0.000,C 90.000,E1 25.463} C_DIS
LIN {X 0.115,Y -555.190,Z 1272.938,A 0.000,B 0.000,C 90.000,E1 24.771} C_DIS
LIN {X 0.180,Y -550.942,Z 1272.935,A 0.000,B 0.000,C 90.000,E1 24.207} C_DIS
LIN {X 0.094,Y -545.252,Z 1272.931,A 0.000,B 0.000,C 90.000,E1 23.515} C_DIS
LIN {X -0.178,Y -537.950,Z 1272.926,A 0.000,B 0.000,C 90.000,E1 22.695} C_DIS
LIN {X 0.028,Y -527.931,Z 1272.920,A 0.000,B 0.000,C 90.000,E1 21.589} C_DIS
LIN {X -0.171,Y -518.881,Z 1272.915,A 0.000,B 0.000,C 90.000,E1 20.663} C_DIS
LIN {X -0.154,Y -509.966,Z 1272.910,A 0.000,B 0.000,C 90.000,E1 19.758} C_DIS
LIN {X -0.154,Y -503.212,Z 1272.906,A 0.000,B 0.000,C 90.000,E1 19.087} C_DIS
LIN {X 0.107,Y -492.198,Z 1272.900,A 0.000,B 0.000,C 90.000,E1 18.000} C_DIS
LIN {X 0.155,Y -486.490,Z 1272.897,A 0.000,B 0.000,C 90.000,E1 17.457} C_DIS
LIN {X 0.059,Y -477.653,Z 1272.893,A 0.000,B 0.000,C 90.000,E1 16.677} C_DIS
LIN {X 0.185,Y -465.779,Z 1272.887,A 0.000,B 0.000,C 90.000,E1 15.607} C_DIS
LIN {X 0.029,Y -446.709,Z 1272.877,A 0.000,B 0.000,C 90.000,E1 13.883} C_DIS
LIN {X 0.014,Y -423.552,Z 1272.865,A 0.000,B 0.000,C 90.000,E1 11.591} C_DIS
LIN {X 0.086,Y -406.393,Z 1272.854,A 0.000,B 0.000,C 90.000,E1 9.726} C_DIS
LIN {X 0.006,Y -400.702,Z 1272.851,A 0.000,B 0.000,C 90.000,E1 9.095} C_DIS
LIN {X 0.034,Y -398.453,Z 1272.849,A 0.000,B 0.000,C 90.000,E1 8.803} C_DIS
LIN {X 0.122,Y -395.408,Z 1272.846,A 0.000,B 0.000,C 90.000,E1 8.341} C_DIS
LIN {X 0.165,Y -394.906,Z 1272.846,A 0.000,B 0.000,C 90.000,E1 8.219} C_DIS
LIN {X 0.127,Y -394.913,Z 1272.846,A 0.000,B 0.000,C 90.000,E1 8.219} C_DIS
LIN {X 0.009,Y -395.522,Z 1272.845,A 0.000,B 0.000,C 90.000,E1 8.049} C_DIS
LIN {X -0.123,Y -396.423,Z 1272.844,A 0.000,B 0.000,C 90.000,E1 7.936} C_DIS
LIN {X -0.146,Y -398.833,Z 1272.843,A 0.000,B 0.000,C 90.000,E1 7.701} C_DIS
LIN {X -0.001,Y -400.545,Z 1272.842,A 0.000,B 0.000,C 90.000,E1 7.530} C_DIS
LIN {X 0.217,Y -409.910,Z 1272.839,A 0.000,B 0.000,C 90.000,E1 6.947} C_DIS
LIN {X 0.100,Y -416.275,Z 1272.837,A 0.000,B 0.000,C 90.000,E1 6.549} C_DIS
LIN {X -0.097,Y -423.978,Z 1272.833,A 0.000,B 0.000,C 90.000,E1 6.030} C_DIS
LIN {X 0.078,Y -433.407,Z 1272.829,A 0.000,B 0.000,C 90.000,E1 5.277} C_DIS
LIN {X 0.115,Y -442.797,Z 1272.825,A 0.000,B 0.000,C 90.000,E1 4.531} C_DIS
LIN {X -0.100,Y -453.524,Z 1272.820,A 0.000,B 0.000,C 90.000,E1 3.669} C_DIS
LIN {X 0.214,Y -460.876,Z 1272.817,A 0.000,B 0.000,C 90.000,E1 2.980} C_DIS
LIN {X 0.202,Y -466.415,Z 1272.814,A 0.000,B 0.000,C 90.000,E1 2.465} C_DIS
LIN {X 0.046,Y -473.351,Z 1272.810,A 0.000,B 0.000,C 90.000,E1 1.776} C_DIS
LIN {X -0.058,Y -478.770,Z 1272.807,A 0.000,B 0.000,C 90.000,E1 1.203} C_DIS
LIN {X -0.022,Y -486.496,Z 1272.802,A 0.000,B 0.000,C 90.000,E1 0.286} C_DIS
LIN {X 0.022,Y -492.622,Z 1272.797,A 0.000,B 0.000,C 90.000,E1 359.484} C_DIS
LIN {X -0.100,Y -497.970,Z 1272.793,A 0.000,B 0.000,C 90.000,E1 358.740} C_DIS
LIN {X 0.031,Y -503.847,Z 1272.788,A 0.000,B 0.000,C 90.000,E1 357.822} C_DIS
LIN {X -0.195,Y -507.541,Z 1272.785,A 0.000,B 0.000,C 90.000,E1 357.249} C_DIS
LIN {X -0.163,Y -511.865,Z 1272.781,A 0.000,B 0.000,C 90.000,E1 356.502} C_DIS
LIN {X -0.086,Y -515.908,Z 1272.776,A 0.000,B 0.000,C 90.000,E1 355.755} C_DIS
LIN {X -0.196,Y -518.915,Z 1272.773,A 0.000,B 0.000,C 90.000,E1 355.179} C_DIS
LIN {X -0.053,Y -522.443,Z 1272.769,A 0.000,B 0.000,C 90.000,E1 354.432} C_DIS
LIN {X 0.130,Y -527.029,Z 1272.763,A 0.000,B 0.000,C 90.000,E1 353.394} C_DIS
LIN {X -0.160,Y -531.018,Z 1272.758,A 0.000,B 0.000,C 90.000,E1 352.413} C_DIS
LIN {X -0.128,Y -534.184,Z 1272.753,A 0.000,B 0.000,C 90.000,E1 351.546} C_DIS
LIN {X -0.065,Y -537.037,Z 1272.748,A 0.000,B 0.000,C 90.000,E1 350.679} C_DIS
LIN {X 0.118,Y -539.589,Z 1272.743,A 0.000,B 0.000,C 90.000,E1 349.803} C_DIS
LIN {X -0.224,Y -542.770,Z 1272.737,A 0.000,B 0.000,C 90.000,E1 348.701} C_DIS
LIN {X 0.023,Y -544.792,Z 1272.732,A 0.000,B 0.000,C 90.000,E1 347.825} C_DIS
LIN {X -0.026,Y -547.282,Z 1272.726,A 0.000,B 0.000,C 90.000,E1 346.700} C_DIS
LIN {X -0.264,Y -548.913,Z 1272.721,A 0.000,B 0.000,C 90.000,E1 345.880} C_DIS
LIN {X 0.178,Y -550.425,Z 1272.717,A 0.000,B 0.000,C 90.000,E1 344.991} C_DIS
LIN {X -0.055,Y -552.439,Z 1272.709,A 0.000,B 0.000,C 90.000,E1 343.614} C_DIS
LIN {X -0.100,Y -553.404,Z 1272.704,A 0.000,B 0.000,C 90.000,E1 342.779} C_DIS
LIN {X 0.280,Y -553.954,Z 1272.701,A 0.000,B 0.000,C 90.000,E1 342.181} C_DIS
LIN {X -0.285,Y -554.491,Z 1272.697,A 0.000,B 0.000,C 90.000,E1 341.402} C_DIS
LIN {X -0.144,Y -554.806,Z 1272.692,A 0.000,B 0.000,C 90.000,E1 340.550} C_DIS
LIN {X -0.283,Y -554.823,Z 1272.689,A 0.000,B 0.000,C 90.000,E1 340.007} C_DIS
LIN {X 0.058,Y -554.551,Z 1272.684,A 0.000,B 0.000,C 90.000,E1 339.135} C_DIS
LIN {X -0.028,Y -553.710,Z 1272.678,A 0.000,B 0.000,C 90.000,E1 338.028} C_DIS
LIN {X -0.183,Y -553.097,Z 1272.675,A 0.000,B 0.000,C 90.000,E1 337.486} C_DIS
LIN {X -0.085,Y -551.412,Z 1272.669,A 0.000,B 0.000,C 90.000,E1 336.357} C_DIS
LIN {X -0.245,Y -548.815,Z 1272.661,A 0.000,B 0.000,C 90.000,E1 334.973} C_DIS
LIN {X 0.028,Y -546.732,Z 1272.656,A 0.000,B 0.000,C 90.000,E1 334.101} C_DIS
LIN {X 0.025,Y -544.397,Z 1272.651,A 0.000,B 0.000,C 90.000,E1 333.256} C_DIS
LIN {X 0.003,Y -541.694,Z 1272.647,A 0.000,B 0.000,C 90.000,E1 332.410} C_DIS
LIN {X -0.045,Y -538.461,Z 1272.642,A 0.000,B 0.000,C 90.000,E1 331.563} C_DIS
LIN {X 0.010,Y -535.400,Z 1272.638,A 0.000,B 0.000,C 90.000,E1 330.845} C_DIS
LIN {X -0.113,Y -531.176,Z 1272.633,A 0.000,B 0.000,C 90.000,E1 329.999} C_DIS
LIN {X -0.019,Y -526.217,Z 1272.629,A 0.000,B 0.000,C 90.000,E1 329.125} C_DIS
LIN {X -0.100,Y -516.698,Z 1272.620,A 0.000,B 0.000,C 90.000,E1 327.533} C_DIS
LIN {X 0.010,Y -512.288,Z 1272.615,A 0.000,B 0.000,C 90.000,E1 326.786} C_DIS
LIN {X -0.017,Y -507.194,Z 1272.610,A 0.000,B 0.000,C 90.000,E1 325.754} C_DIS
LIN {X -0.115,Y -505.919,Z 1272.608,A 0.000,B 0.000,C 90.000,E1 325.468} C_DIS
LIN {X -0.006,Y -503.991,Z 1272.605,A 0.000,B 0.000,C 90.000,E1 324.895} C_DIS
LIN {X 0.188,Y -502.449,Z 1272.602,A 0.000,B 0.000,C 90.000,E1 324.276} C_DIS
LIN {X -0.156,Y -500.779,Z 1272.597,A 0.000,B 0.000,C 90.000,E1 323.417} C_DIS
LIN {X 0.185,Y -499.913,Z 1272.592,A 0.000,B 0.000,C 90.000,E1 322.477} C_DIS
LIN {X -0.251,Y -499.304,Z 1272.582,A 0.000,B 0.000,C 90.000,E1 320.723} C_DIS
LIN {X 0.014,Y -499.621,Z 1272.568,A 0.000,B 0.000,C 90.000,E1 318.286} C_DIS
LIN {X 0.009,Y -499.931,Z 1272.560,A 0.000,B 0.000,C 90.000,E1 316.782} C_DIS
LIN {X -0.026,Y -500.157,Z 1272.552,A 0.000,B 0.000,C 90.000,E1 315.283} C_DIS
LIN {X -0.057,Y -500.467,Z 1272.543,A 0.000,B 0.000,C 90.000,E1 313.785} C_DIS
LIN {X -0.006,Y -500.912,Z 1272.532,A 0.000,B 0.000,C 90.000,E1 311.676} C_DIS
LIN {X -0.057,Y -501.070,Z 1272.527,A 0.000,B 0.000,C 90.000,E1 310.782} C_DIS
LIN {X -0.072,Y -501.349,Z 1272.513,A 0.000,B 0.000,C 90.000,E1 308.382} C_DIS
LIN {X -0.080,Y -501.666,Z 1272.503,A 0.000,B 0.000,C 90.000,E1 306.583} C_DIS
LIN {X -0.026,Y -501.831,Z 1272.498,A 0.000,B 0.000,C 90.000,E1 305.678} C_DIS
LIN {X 0.095,Y -501.868,Z 1272.488,A 0.000,B 0.000,C 90.000,E1 303.865} C_DIS
LIN {X 0.327,Y -501.652,Z 1272.480,A 0.000,B 0.000,C 90.000,E1 302.339} C_DIS
LIN {X 0.107,Y -501.493,Z 1272.475,A 0.000,B 0.000,C 90.000,E1 301.465} C_DIS
LIN {X -0.116,Y -501.011,Z 1272.470,A 0.000,B 0.000,C 90.000,E1 300.590} C_DIS
LIN {X 0.088,Y -500.281,Z 1272.465,A 0.000,B 0.000,C 90.000,E1 299.667} C_DIS
LIN {X 0.281,Y -499.210,Z 1272.460,A 0.000,B 0.000,C 90.000,E1 298.743} C_DIS
LIN {X 0.176,Y -498.076,Z 1272.457,A 0.000,B 0.000,C 90.000,E1 298.153} C_DIS
LIN {X -0.215,Y -497.294,Z 1272.455,A 0.000,B 0.000,C 90.000,E1 297.897} C_DIS
LIN {X -0.167,Y -496.196,Z 1272.453,A 0.000,B 0.000,C 90.000,E1 297.590} C_DIS
LIN {X 0.093,Y -483.286,Z 1272.436,A 0.000,B 0.000,C 90.000,E1 294.515} C_DIS
LIN {X 0.174,Y -472.175,Z 1272.419,A 0.000,B 0.000,C 90.000,E1 291.408} C_DIS
LIN {X 0.167,Y -461.928,Z 1272.400,A 0.000,B 0.000,C 90.000,E1 287.946} C_DIS
LIN {X 0.101,Y -453.009,Z 1272.379,A 0.000,B 0.000,C 90.000,E1 284.120} C_DIS
LIN {X -0.096,Y -445.464,Z 1272.353,A 0.000,B 0.000,C 90.000,E1 279.613} C_DIS
LIN {X -0.002,Y -439.989,Z 1272.319,A 0.000,B 0.000,C 90.000,E1 273.383} C_DIS
LIN {X -0.055,Y -442.897,Z 1272.260,A 0.000,B 0.000,C 90.000,E1 262.875} C_DIS
LIN {X -0.115,Y -449.553,Z 1272.233,A 0.000,B 0.000,C 90.000,E1 257.993} C_DIS
LIN {X -0.047,Y -458.157,Z 1272.210,A 0.000,B 0.000,C 90.000,E1 253.795} C_DIS
LIN {X -0.046,Y -467.576,Z 1272.191,A 0.000,B 0.000,C 90.000,E1 250.296} C_DIS
LIN {X 0.120,Y -469.438,Z 1272.187,A 0.000,B 0.000,C 90.000,E1 249.645} C_DIS
LIN {X 0.069,Y -470.022,Z 1272.185,A 0.000,B 0.000,C 90.000,E1 249.337} C_DIS
LIN {X -0.024,Y -470.753,Z 1272.182,A 0.000,B 0.000,C 90.000,E1 248.720} C_DIS
LIN {X -0.110,Y -471.203,Z 1272.178,A 0.000,B 0.000,C 90.000,E1 248.103} C_DIS
LIN {X -0.233,Y -471.342,Z 1272.173,A 0.000,B 0.000,C 90.000,E1 247.177} C_DIS
LIN {X -0.169,Y -471.221,Z 1272.168,A 0.000,B 0.000,C 90.000,E1 246.230} C_DIS
LIN {X -0.099,Y -470.864,Z 1272.163,A 0.000,B 0.000,C 90.000,E1 245.281} C_DIS
LIN {X 0.075,Y -469.924,Z 1272.154,A 0.000,B 0.000,C 90.000,E1 243.691} C_DIS
LIN {X -0.033,Y -468.779,Z 1272.143,A 0.000,B 0.000,C 90.000,E1 241.820} C_DIS
LIN {X 0.053,Y -467.796,Z 1272.133,A 0.000,B 0.000,C 90.000,E1 239.921} C_DIS
LIN {X -0.054,Y -466.597,Z 1272.122,A 0.000,B 0.000,C 90.000,E1 238.043} C_DIS
LIN {X -0.044,Y -464.802,Z 1272.108,A 0.000,B 0.000,C 90.000,E1 235.515} C_DIS
LIN {X 0.055,Y -463.329,Z 1272.094,A 0.000,B 0.000,C 90.000,E1 232.970} C_DIS
LIN {X 0.012,Y -462.171,Z 1272.080,A 0.000,B 0.000,C 90.000,E1 230.436} C_DIS
LIN {X -0.237,Y -461.365,Z 1272.068,A 0.000,B 0.000,C 90.000,E1 228.243} C_DIS
LIN {X 0.110,Y -460.687,Z 1272.056,A 0.000,B 0.000,C 90.000,E1 225.972} C_DIS
LIN {X -0.223,Y -460.143,Z 1272.043,A 0.000,B 0.000,C 90.000,E1 223.785} C_DIS
LIN {X 0.018,Y -460.223,Z 1272.022,A 0.000,B 0.000,C 90.000,E1 219.930} C_DIS
LIN {X 0.168,Y -461.579,Z 1272.001,A 0.000,B 0.000,C 90.000,E1 216.091} C_DIS
LIN {X -0.189,Y -464.168,Z 1271.983,A 0.000,B 0.000,C 90.000,E1 212.959} C_DIS
LIN {X -0.066,Y -467.034,Z 1271.969,A 0.000,B 0.000,C 90.000,E1 210.413} C_DIS
LIN {X 0.225,Y -469.293,Z 1271.958,A 0.000,B 0.000,C 90.000,E1 208.487} C_DIS
LIN {X -0.242,Y -472.719,Z 1271.943,A 0.000,B 0.000,C 90.000,E1 205.720} C_DIS
LIN {X -0.114,Y -476.389,Z 1271.929,A 0.000,B 0.000,C 90.000,E1 203.206} C_DIS
LIN {X 0.197,Y -481.448,Z 1271.912,A 0.000,B 0.000,C 90.000,E1 200.066} C_DIS
LIN {X 0.033,Y -484.787,Z 1271.901,A 0.000,B 0.000,C 90.000,E1 198.236} C_DIS
LIN {X 0.113,Y -488.834,Z 1271.889,A 0.000,B 0.000,C 90.000,E1 196.079} C_DIS
LIN {X 0.058,Y -493.482,Z 1271.876,A 0.000,B 0.000,C 90.000,E1 193.647} C_DIS
LIN {X 0.080,Y -497.153,Z 1271.866,A 0.000,B 0.000,C 90.000,E1 191.827} C_DIS
LIN {X 0.084,Y -500.768,Z 1271.856,A 0.000,B 0.000,C 90.000,E1 190.018} C_DIS
LIN {X 0.079,Y -504.411,Z 1271.846,A 0.000,B 0.000,C 90.000,E1 188.219} C_DIS
LIN {X 0.142,Y -507.563,Z 1271.838,A 0.000,B 0.000,C 90.000,E1 186.720} C_DIS
LIN {X -0.242,Y -510.550,Z 1271.829,A 0.000,B 0.000,C 90.000,E1 185.277} C_DIS
LIN {X -0.198,Y -514.144,Z 1271.819,A 0.000,B 0.000,C 90.000,E1 183.498} C_DIS
LIN {X -0.028,Y -517.015,Z 1271.811,A 0.000,B 0.000,C 90.000,E1 182.007} C_DIS
LIN {X 0.195,Y -519.751,Z 1271.803,A 0.000,B 0.000,C 90.000,E1 180.516} C_DIS
LIN {X -0.111,Y -522.943,Z 1271.793,A 0.000,B 0.000,C 90.000,E1 178.797} C_DIS
LIN {X 0.258,Y -524.916,Z 1271.787,A 0.000,B 0.000,C 90.000,E1 177.593} C_DIS
LIN {X 0.138,Y -526.803,Z 1271.780,A 0.000,B 0.000,C 90.000,E1 176.445} C_DIS
LIN {X 0.048,Y -528.854,Z 1271.772,A 0.000,B 0.000,C 90.000,E1 175.008} C_DIS
LIN {X 0.022,Y -530.280,Z 1271.766,A 0.000,B 0.000,C 90.000,E1 173.856} C_DIS
LIN {X -0.018,Y -531.218,Z 1271.761,A 0.000,B 0.000,C 90.000,E1 172.996} C_DIS
LIN {X 0.089,Y -532.505,Z 1271.753,A 0.000,B 0.000,C 90.000,E1 171.546} C_DIS
LIN {X 0.134,Y -533.159,Z 1271.748,A 0.000,B 0.000,C 90.000,E1 170.679} C_DIS
LIN {X -0.202,Y -533.793,Z 1271.742,A 0.000,B 0.000,C 90.000,E1 169.567} C_DIS
LIN {X -0.103,Y -534.230,Z 1271.736,A 0.000,B 0.000,C 90.000,E1 168.409} C_DIS
LIN {X 0.214,Y -534.471,Z 1271.729,A 0.000,B 0.000,C 90.000,E1 167.229} C_DIS
LIN {X 0.127,Y -534.599,Z 1271.720,A 0.000,B 0.000,C 90.000,E1 165.519} C_DIS
LIN {X 0.178,Y -535.094,Z 1271.702,A 0.000,B 0.000,C 90.000,E1 162.362} C_DIS
LIN {X 0.143,Y -535.737,Z 1271.696,A 0.000,B 0.000,C 90.000,E1 161.221} C_DIS
LIN {X 0.293,Y -536.900,Z 1271.689,A 0.000,B 0.000,C 90.000,E1 160.061} C_DIS
LIN {X 0.246,Y -538.268,Z 1271.685,A 0.000,B 0.000,C 90.000,E1 159.209} C_DIS
LIN {X -0.292,Y -540.085,Z 1271.680,A 0.000,B 0.000,C 90.000,E1 158.411} C_DIS
LIN {X -0.110,Y -542.514,Z 1271.675,A 0.000,B 0.000,C 90.000,E1 157.539} C_DIS
LIN {X 0.104,Y -545.519,Z 1271.671,A 0.000,B 0.000,C 90.000,E1 156.666} C_DIS
LIN {X -0.146,Y -549.275,Z 1271.666,A 0.000,B 0.000,C 90.000,E1 155.845} C_DIS
LIN {X -0.120,Y -552.245,Z 1271.663,A 0.000,B 0.000,C 90.000,E1 155.281} C_DIS
LIN {X 0.101,Y -558.251,Z 1271.657,A 0.000,B 0.000,C 90.000,E1 154.280} C_DIS
LIN {X -0.049,Y -566.959,Z 1271.650,A 0.000,B 0.000,C 90.000,E1 153.050} C_DIS
LIN {X 0.239,Y -579.907,Z 1271.641,A 0.000,B 0.000,C 90.000,E1 151.385} C_DIS
LIN {X 0.111,Y -586.336,Z 1271.637,A 0.000,B 0.000,C 90.000,E1 150.589} C_DIS
LIN {X 0.124,Y -592.623,Z 1271.632,A 0.000,B 0.000,C 90.000,E1 149.793} C_DIS
LIN {X 0.129,Y -598.606,Z 1271.628,A 0.000,B 0.000,C 90.000,E1 148.997} C_DIS
LIN {X 0.118,Y -606.123,Z 1271.622,A 0.000,B 0.000,C 90.000,E1 147.946} C_DIS
LIN {X -0.205,Y -609.775,Z 1271.619,A 0.000,B 0.000,C 90.000,E1 147.454} C_DIS
LIN {X 0.013,Y -613.157,Z 1271.616,A 0.000,B 0.000,C 90.000,E1 146.914} C_DIS
LIN {X 0.003,Y -619.588,Z 1271.610,A 0.000,B 0.000,C 90.000,E1 145.881} C_DIS
LIN {X -0.225,Y -622.474,Z 1271.608,A 0.000,B 0.000,C 90.000,E1 145.388} C_DIS
LIN {X 0.041,Y -626.538,Z 1271.603,A 0.000,B 0.000,C 90.000,E1 144.609} C_DIS
LIN {X -0.036,Y -630.347,Z 1271.599,A 0.000,B 0.000,C 90.000,E1 143.863} C_DIS
LIN {X 0.180,Y -632.782,Z 1271.596,A 0.000,B 0.000,C 90.000,E1 143.336} C_DIS
LIN {X -0.093,Y -636.105,Z 1271.592,A 0.000,B 0.000,C 90.000,E1 142.603} C_DIS
LIN {X 0.059,Y -641.013,Z 1271.585,A 0.000,B 0.000,C 90.000,E1 141.331} C_DIS
LIN {X 0.361,Y -642.808,Z 1271.583,A 0.000,B 0.000,C 90.000,E1 140.803} C_DIS
LIN {X 0.101,Y -646.256,Z 1271.577,A 0.000,B 0.000,C 90.000,E1 139.828} C_DIS
LIN {X 0.250,Y -650.977,Z 1271.569,A 0.000,B 0.000,C 90.000,E1 138.324} C_DIS
LIN {X -0.396,Y -654.034,Z 1271.563,A 0.000,B 0.000,C 90.000,E1 137.391} C_DIS
LIN {X -0.115,Y -657.556,Z 1271.556,A 0.000,B 0.000,C 90.000,E1 136.134} C_DIS
LIN {X -0.265,Y -661.991,Z 1271.548,A 0.000,B 0.000,C 90.000,E1 134.676} C_DIS
LIN {X 0.152,Y -666.533,Z 1271.540,A 0.000,B 0.000,C 90.000,E1 133.176} C_DIS
LIN {X -0.288,Y -671.073,Z 1271.532,A 0.000,B 0.000,C 90.000,E1 131.757} C_DIS
LIN {X -0.153,Y -675.389,Z 1271.524,A 0.000,B 0.000,C 90.000,E1 130.297} C_DIS
LIN {X 0.122,Y -678.861,Z 1271.517,A 0.000,B 0.000,C 90.000,E1 129.072} C_DIS
LIN {X -0.064,Y -682.237,Z 1271.510,A 0.000,B 0.000,C 90.000,E1 127.890} C_DIS
LIN {X -0.040,Y -685.986,Z 1271.503,A 0.000,B 0.000,C 90.000,E1 126.457} C_DIS
LIN {X 0.048,Y -689.413,Z 1271.495,A 0.000,B 0.000,C 90.000,E1 125.025} C_DIS
LIN {X 0.125,Y -691.584,Z 1271.489,A 0.000,B 0.000,C 90.000,E1 124.072} C_DIS
LIN {X 0.263,Y -693.971,Z 1271.483,A 0.000,B 0.000,C 90.000,E1 122.880} C_DIS
LIN {X 0.049,Y -696.224,Z 1271.476,A 0.000,B 0.000,C 90.000,E1 121.720} C_DIS
LIN {X 0.104,Y -698.289,Z 1271.470,A 0.000,B 0.000,C 90.000,E1 120.541} C_DIS
LIN {X -0.137,Y -700.418,Z 1271.462,A 0.000,B 0.000,C 90.000,E1 119.155} C_DIS
LIN {X -0.279,Y -701.612,Z 1271.457,A 0.000,B 0.000,C 90.000,E1 118.231} C_DIS
LIN {X -0.070,Y -702.388,Z 1271.453,A 0.000,B 0.000,C 90.000,E1 117.513} C_DIS
LIN {X 0.141,Y -702.848,Z 1271.449,A 0.000,B 0.000,C 90.000,E1 116.796} C_DIS
LIN {X 0.042,Y -703.048,Z 1271.445,A 0.000,B 0.000,C 90.000,E1 116.104} C_DIS
LIN {X -0.029,Y -703.004,Z 1271.443,A 0.000,B 0.000,C 90.000,E1 115.643} C_DIS
LIN {X -0.126,Y -702.598,Z 1271.439,A 0.000,B 0.000,C 90.000,E1 114.951} C_DIS
LIN {X -0.141,Y -702.422,Z 1271.437,A 0.000,B 0.000,C 90.000,E1 114.719} C_DIS
LIN {X -0.223,Y -701.720,Z 1271.435,A 0.000,B 0.000,C 90.000,E1 114.259} C_DIS
LIN {X -0.234,Y -701.218,Z 1271.433,A 0.000,B 0.000,C 90.000,E1 114.027} C_DIS
LIN {X 0.312,Y -699.390,Z 1271.431,A 0.000,B 0.000,C 90.000,E1 113.515} C_DIS
LIN {X -0.196,Y -698.836,Z 1271.430,A 0.000,B 0.000,C 90.000,E1 113.439} C_DIS
LIN {X -0.208,Y -696.983,Z 1271.429,A 0.000,B 0.000,C 90.000,E1 113.206} C_DIS
LIN {X 0.175,Y -693.956,Z 1271.427,A 0.000,B 0.000,C 90.000,E1 112.823} C_DIS
LIN {X 0.030,Y -692.451,Z 1271.426,A 0.000,B 0.000,C 90.000,E1 112.717} C_DIS
LIN {X 0.123,Y -688.227,Z 1271.425,A 0.000,B 0.000,C 90.000,E1 112.514} C_DIS
LIN {X -0.029,Y -682.683,Z 1271.424,A 0.000,B 0.000,C 90.000,E1 112.333} C_DIS
LIN {X 0.115,Y -678.274,Z 1271.423,A 0.000,B 0.000,C 90.000,E1 112.206} C_DIS
LIN {X -0.130,Y -670.063,Z 1271.423,A 0.000,B 0.000,C 90.000,E1 112.153} C_DIS
LIN {X -0.167,Y -636.169,Z 1271.423,A 0.000,B 0.000,C 90.000,E1 112.153} C_DIS
LIN {X 0.066,Y -632.890,Z 1271.422,A 0.000,B 0.000,C 90.000,E1 112.025} C_DIS
LIN {X 0.024,Y -632.751,Z 1271.422,A 0.000,B 0.000,C 90.000,E1 112.025} C_DIS
LIN {X -0.174,Y -633.081,Z 1271.422,A 0.000,B 0.000,C 90.000,E1 111.897} C_DIS
LIN {X -0.160,Y -633.549,Z 1271.421,A 0.000,B 0.000,C 90.000,E1 111.770} C_DIS
LIN {X 0.247,Y -635.587,Z 1271.419,A 0.000,B 0.000,C 90.000,E1 111.354} C_DIS
LIN {X 0.224,Y -643.024,Z 1271.413,A 0.000,B 0.000,C 90.000,E1 110.301} C_DIS
LIN {X -0.079,Y -647.051,Z 1271.409,A 0.000,B 0.000,C 90.000,E1 109.704} C_DIS
LIN {X -0.272,Y -651.746,Z 1271.405,A 0.000,B 0.000,C 90.000,E1 108.852} C_DIS
LIN {X -0.293,Y -654.858,Z 1271.401,A 0.000,B 0.000,C 90.000,E1 108.236} C_DIS
LIN {X 0.167,Y -658.257,Z 1271.397,A 0.000,B 0.000,C 90.000,E1 107.457} C_DIS
LIN {X 0.033,Y -661.375,Z 1271.393,A 0.000,B 0.000,C 90.000,E1 106.732} C_DIS
LIN {X -0.167,Y -663.341,Z 1271.390,A 0.000,B 0.000,C 90.000,E1 106.260} C_DIS
LIN {X 0.381,Y -665.851,Z 1271.386,A 0.000,B 0.000,C 90.000,E1 105.481} C_DIS
LIN {X 0.214,Y -667.273,Z 1271.384,A 0.000,B 0.000,C 90.000,E1 105.009} C_DIS
LIN {X 0.057,Y -668.489,Z 1271.381,A 0.000,B 0.000,C 90.000,E1 104.537} C_DIS
LIN {X -0.161,Y -669.873,Z 1271.377,A 0.000,B 0.000,C 90.000,E1 103.828} C_DIS
LIN {X -0.300,Y -670.586,Z 1271.374,A 0.000,B 0.000,C 90.000,E1 103.355} C_DIS
LIN {X 0.151,Y -671.155,Z 1271.370,A 0.000,B 0.000,C 90.000,E1 102.591} C_DIS
LIN {X 0.018,Y -671.382,Z 1271.367,A 0.000,B 0.000,C 90.000,E1 102.119} C_DIS
LIN {X -0.317,Y -671.138,Z 1271.363,A 0.000,B 0.000,C 90.000,E1 101.422} C_DIS
LIN {X 0.206,Y -670.802,Z 1271.361,A 0.000,B 0.000,C 90.000,E1 100.894} C_DIS
LIN {X -0.057,Y -670.235,Z 1271.358,A 0.000,B 0.000,C 90.000,E1 100.433} C_DIS
LIN {X -0.202,Y -669.404,Z 1271.355,A 0.000,B 0.000,C 90.000,E1 99.962} C_DIS
LIN {X 0.191,Y -668.320,Z 1271.353,A 0.000,B 0.000,C 90.000,E1 99.443} C_DIS
LIN {X 0.027,Y -666.898,Z 1271.350,A 0.000,B 0.000,C 90.000,E1 98.973} C_DIS
LIN {X -0.162,Y -666.087,Z 1271.349,A 0.000,B 0.000,C 90.000,E1 98.746} C_DIS
LIN {X 0.312,Y -664.175,Z 1271.346,A 0.000,B 0.000,C 90.000,E1 98.219} C_DIS
LIN {X -0.079,Y -661.311,Z 1271.343,A 0.000,B 0.000,C 90.000,E1 97.644} C_DIS
LIN {X 0.265,Y -658.652,Z 1271.340,A 0.000,B 0.000,C 90.000,E1 97.125} C_DIS
LIN {X -0.090,Y -654.848,Z 1271.336,A 0.000,B 0.000,C 90.000,E1 96.543} C_DIS
LIN {X 0.137,Y -651.458,Z 1271.334,A 0.000,B 0.000,C 90.000,E1 96.030} C_DIS
LIN {X -0.284,Y -646.596,Z 1271.330,A 0.000,B 0.000,C 90.000,E1 95.448} C_DIS
LIN {X -0.103,Y -642.347,Z 1271.327,A 0.000,B 0.000,C 90.000,E1 94.935} C_DIS
LIN {X 0.107,Y -637.715,Z 1271.325,A 0.000,B 0.000,C 90.000,E1 94.416} C_DIS
LIN {X 0.287,Y -631.444,Z 1271.321,A 0.000,B 0.000,C 90.000,E1 93.784} C_DIS
LIN {X 0.042,Y -626.259,Z 1271.319,A 0.000,B 0.000,C 90.000,E1 93.326} C_DIS
LIN {X 0.109,Y -619.374,Z 1271.315,A 0.000,B 0.000,C 90.000,E1 92.751} C_DIS
LIN {X -0.291,Y -613.710,Z 1271.313,A 0.000,B 0.000,C 90.000,E1 92.350} C_DIS
LIN {X 0.001,Y -607.840,Z 1271.311,A 0.000,B 0.000,C 90.000,E1 91.892} C_DIS
LIN {X -0.155,Y -601.787,Z 1271.308,A 0.000,B 0.000,C 90.000,E1 91.489} C_DIS
LIN {X -0.039,Y -595.430,Z 1271.306,A 0.000,B 0.000,C 90.000,E1 91.088} C_DIS
LIN {X -0.161,Y -588.731,Z 1271.304,A 0.000,B 0.000,C 90.000,E1 90.745} C_DIS
LIN {X 0.239,Y -581.653,Z 1271.302,A 0.000,B 0.000,C 90.000,E1 90.401} C_DIS
LIN {X -0.080,Y -576.393,Z 1271.301,A 0.000,B 0.000,C 90.000,E1 90.229} C_DIS
LIN {X 0.230,Y -572.200,Z 1271.300,A 0.000,B 0.000,C 90.000,E1 90.000} C_DIS
LIN {X -0.097,Y -568.873,Z 1271.298,A 0.000,B 0.000,C 90.000,E1 89.656} C_DIS
LIN {X -0.139,Y -568.859,Z 1271.298,A 0.000,B 0.000,C 90.000,E1 89.656} C_DIS
LIN {X -0.152,Y -568.485,Z 1271.297,A 0.000,B 0.000,C 90.000,E1 89.427} C_DIS
LIN {X 0.096,Y -568.520,Z 1271.294,A 0.000,B 0.000,C 90.000,E1 88.854} C_DIS
LIN {X 0.129,Y -570.460,Z 1271.280,A 0.000,B 0.000,C 90.000,E1 86.388} C_DIS
LIN {X -0.131,Y -573.234,Z 1271.265,A 0.000,B 0.000,C 90.000,E1 83.685} C_DIS
LIN {X 0.120,Y -574.685,Z 1271.257,A 0.000,B 0.000,C 90.000,E1 82.299} C_DIS
LIN {X 0.276,Y -575.935,Z 1271.251,A 0.000,B 0.000,C 90.000,E1 81.197} C_DIS
LIN {X -0.118,Y -577.101,Z 1271.245,A 0.000,B 0.000,C 90.000,E1 80.151} C_DIS
LIN {X 0.068,Y -578.144,Z 1271.239,A 0.000,B 0.000,C 90.000,E1 79.050} C_DIS
LIN {X -0.093,Y -579.729,Z 1271.229,A 0.000,B 0.000,C 90.000,E1 77.173} C_DIS
LIN {X -0.331,Y -580.558,Z 1271.223,A 0.000,B 0.000,C 90.000,E1 76.117} C_DIS
LIN {X -0.193,Y -581.524,Z 1271.215,A 0.000,B 0.000,C 90.000,E1 74.755} C_DIS
LIN {X 0.119,Y -582.296,Z 1271.208,A 0.000,B 0.000,C 90.000,E1 73.378} C_DIS
LIN {X 0.112,Y -583.338,Z 1271.199,A 0.000,B 0.000,C 90.000,E1 71.764} C_DIS
LIN {X -0.253,Y -584.240,Z 1271.190,A 0.000,B 0.000,C 90.000,E1 70.188} C_DIS
LIN {X -0.117,Y -585.449,Z 1271.178,A 0.000,B 0.000,C 90.000,E1 68.028} C_DIS
LIN {X -0.068,Y -587.297,Z 1271.165,A 0.000,B 0.000,C 90.000,E1 65.613} C_DIS
LIN {X -0.223,Y -588.553,Z 1271.156,A 0.000,B 0.000,C 90.000,E1 64.024} C_DIS
LIN {X -0.191,Y -590.155,Z 1271.145,A 0.000,B 0.000,C 90.000,E1 62.153} C_DIS
LIN {X -0.023,Y -591.694,Z 1271.136,A 0.000,B 0.000,C 90.000,E1 60.539} C_DIS
LIN {X 0.049,Y -593.109,Z 1271.129,A 0.000,B 0.000,C 90.000,E1 59.203} C_DIS
LIN {X 0.359,Y -594.781,Z 1271.120,A 0.000,B 0.000,C 90.000,E1 57.582} C_DIS
LIN {X 0.204,Y -596.378,Z 1271.111,A 0.000,B 0.000,C 90.000,E1 56.008} C_DIS
LIN {X 0.069,Y -597.920,Z 1271.103,A 0.000,B 0.000,C 90.000,E1 54.436} C_DIS
LIN {X 0.170,Y -599.248,Z 1271.094,A 0.000,B 0.000,C 90.000,E1 52.844} C_DIS
LIN {X 0.307,Y -600.488,Z 1271.085,A 0.000,B 0.000,C 90.000,E1 51.251} C_DIS
LIN {X -0.032,Y -601.271,Z 1271.079,A 0.000,B 0.000,C 90.000,E1 50.231} C_DIS
LIN {X 0.022,Y -601.699,Z 1271.073,A 0.000,B 0.000,C 90.000,E1 49.175} C_DIS
LIN {X 0.070,Y -602.380,Z 1271.064,A 0.000,B 0.000,C 90.000,E1 47.595} C_DIS
LIN {X 0.136,Y -602.760,Z 1271.059,A 0.000,B 0.000,C 90.000,E1 46.539} C_DIS
LIN {X 0.181,Y -602.973,Z 1271.053,A 0.000,B 0.000,C 90.000,E1 45.486} C_DIS
LIN {X 0.230,Y -602.925,Z 1271.047,A 0.000,B 0.000,C 90.000,E1 44.433} C_DIS
LIN {X 0.072,Y -602.688,Z 1271.040,A 0.000,B 0.000,C 90.000,E1 43.137} C_DIS
LIN {X -0.272,Y -602.130,Z 1271.031,A 0.000,B 0.000,C 90.000,E1 41.595} C_DIS
LIN {X -0.206,Y -601.666,Z 1271.025,A 0.000,B 0.000,C 90.000,E1 40.539} C_DIS
LIN {X -0.174,Y -601.472,Z 1271.022,A 0.000,B 0.000,C 90.000,E1 40.011} C_DIS
LIN {X -0.120,Y -600.838,Z 1271.016,A 0.000,B 0.000,C 90.000,E1 38.955} C_DIS
LIN {X 0.019,Y -600.129,Z 1271.011,A 0.000,B 0.000,C 90.000,E1 37.890} C_DIS
LIN {X -0.080,Y -598.768,Z 1271.003,A 0.000,B 0.000,C 90.000,E1 36.583} C_DIS
LIN {X 0.037,Y -597.380,Z 1270.997,A 0.000,B 0.000,C 90.000,E1 35.518} C_DIS
LIN {X 0.160,Y -596.616,Z 1270.995,A 0.000,B 0.000,C 90.000,E1 34.978} C_DIS
LIN {X 0.242,Y -594.713,Z 1270.989,A 0.000,B 0.000,C 90.000,E1 33.913} C_DIS
LIN {X -0.253,Y -593.150,Z 1270.984,A 0.000,B 0.000,C 90.000,E1 33.166} C_DIS
LIN {X 0.057,Y -591.236,Z 1270.980,A 0.000,B 0.000,C 90.000,E1 32.339} C_DIS
LIN {X 0.222,Y -588.349,Z 1270.974,A 0.000,B 0.000,C 90.000,E1 31.258} C_DIS
LIN {X 0.167,Y -585.687,Z 1270.969,A 0.000,B 0.000,C 90.000,E1 30.463} C_DIS
LIN {X 0.213,Y -583.761,Z 1270.966,A 0.000,B 0.000,C 90.000,E1 29.922} C_DIS
LIN {X -0.043,Y -581.569,Z 1270.963,A 0.000,B 0.000,C 90.000,E1 29.411} C_DIS
LIN {X -0.309,Y -576.717,Z 1270.957,A 0.000,B 0.000,C 90.000,E1 28.359} C_DIS
LIN {X 0.017,Y -572.368,Z 1270.953,A 0.000,B 0.000,C 90.000,E1 27.513} C_DIS
LIN {X -0.309,Y -569.294,Z 1270.950,A 0.000,B 0.000,C 90.000,E1 27.001} C_DIS
LIN {X 0.108,Y -566.061,Z 1270.947,A 0.000,B 0.000,C 90.000,E1 26.411} C_DIS
LIN {X -0.043,Y -559.766,Z 1270.942,A 0.000,B 0.000,C 90.000,E1 25.463} C_DIS
LIN {X 0.054,Y -555.879,Z 1270.938,A 0.000,B 0.000,C 90.000,E1 24.899} C_DIS
LIN {X 0.014,Y -550.527,Z 1270.935,A 0.000,B 0.000,C 90.000,E1 24.207} C_DIS
LIN {X 0.046,Y -546.000,Z 1270.931,A 0.000,B 0.000,C 90.000,E1 23.643} C_DIS
LIN {X -0.216,Y -538.782,Z 1270.927,A 0.000,B 0.000,C 90.000,E1 22.823} C_DIS
LIN {X 0.094,Y -528.408,Z 1270.920,A 0.000,B 0.000,C 90.000,E1 21.663} C_DIS
LIN {X -0.202,Y -519.267,Z 1270.915,A 0.000,B 0.000,C 90.000,E1 20.737} C_DIS
LIN {X 0.099,Y -508.641,Z 1270.909,A 0.000,B 0.000,C 90.000,E1 19.631} C_DIS
LIN {X 0.075,Y -499.331,Z 1270.904,A 0.000,B 0.000,C 90.000,E1 18.725} C_DIS
LIN {X -0.195,Y -490.830,Z 1270.900,A 0.000,B 0.000,C 90.000,E1 17.946} C_DIS
LIN {X -0.029,Y -485.172,Z 1270.897,A 0.000,B 0.000,C 90.000,E1 17.402} C_DIS
LIN {X 0.073,Y -477.881,Z 1270.893,A 0.000,B 0.000,C 90.000,E1 16.732} C_DIS
LIN {X 0.245,Y -466.026,Z 1270.887,A 0.000,B 0.000,C 90.000,E1 15.662} C_DIS
LIN {X -0.130,Y -445.477,Z 1270.877,A 0.000,B 0.000,C 90.000,E1 13.828} C_DIS
LIN {X 0.146,Y -422.263,Z 1270.864,A 0.000,B 0.000,C 90.000,E1 11.478} C_DIS
LIN {X 0.162,Y -405.110,Z 1270.854,A 0.000,B 0.000,C 90.000,E1 9.613} C_DIS
LIN {X 0.089,Y -399.533,Z 1270.850,A 0.000,B 0.000,C 90.000,E1 8.973} C_DIS
LIN {X -0.033,Y -395.075,Z 1270.846,A 0.000,B 0.000,C 90.000,E1 8.341} C_DIS
LIN {X 0.075,Y -394.944,Z 1270.846,A 0.000,B 0.000,C 90.000,E1 8.276} C_DIS
LIN {X 0.036,Y -394.958,Z 1270.846,A 0.000,B 0.000,C 90.000,E1 8.276} C_DIS
LIN {X 0.004,Y -395.684,Z 1270.845,A 0.000,B 0.000,C 90.000,E1 8.049} C_DIS
LIN {X -0.215,Y -396.234,Z 1270.844,A 0.000,B 0.000,C 90.000,E1 7.992} C_DIS
LIN {X 0.139,Y -400.503,Z 1270.842,A 0.000,B 0.000,C 90.000,E1 7.530} C_DIS
LIN {X -0.093,Y -411.762,Z 1270.838,A 0.000,B 0.000,C 90.000,E1 6.891} C_DIS
LIN {X 0.156,Y -419.658,Z 1270.835,A 0.000,B 0.000,C 90.000,E1 6.315} C_DIS
LIN {X 0.129,Y -425.990,Z 1270.833,A 0.000,B 0.000,C 90.000,E1 5.853} C_DIS
LIN {X -0.210,Y -435.474,Z 1270.829,A 0.000,B 0.000,C 90.000,E1 5.163} C_DIS
LIN {X -0.100,Y -443.281,Z 1270.825,A 0.000,B 0.000,C 90.000,E1 4.531} C_DIS
LIN {X 0.172,Y -452.562,Z 1270.821,A 0.000,B 0.000,C 90.000,E1 3.726} C_DIS
LIN {X 0.054,Y -460.054,Z 1270.817,A 0.000,B 0.000,C 90.000,E1 3.094} C_DIS
LIN {X 0.137,Y -467.285,Z 1270.813,A 0.000,B 0.000,C 90.000,E1 2.407} C_DIS
LIN {X -0.044,Y -474.227,Z 1270.810,A 0.000,B 0.000,C 90.000,E1 1.718} C_DIS
LIN {X -0.124,Y -479.625,Z 1270.806,A 0.000,B 0.000,C 90.000,E1 1.146} C_DIS
LIN {X -0.054,Y -487.327,Z 1270.801,A 0.000,B 0.000,C 90.000,E1 0.229} C_DIS
LIN {X 0.025,Y -492.967,Z 1270.797,A 0.000,B 0.000,C 90.000,E1 359.484} C_DIS
LIN {X 0.085,Y -499.338,Z 1270.792,A 0.000,B 0.000,C 90.000,E1 358.568} C_DIS
LIN {X 0.040,Y -504.247,Z 1270.788,A 0.000,B 0.000,C 90.000,E1 357.822} C_DIS
LIN {X -0.183,Y -507.966,Z 1270.785,A 0.000,B 0.000,C 90.000,E1 357.249} C_DIS
LIN {X -0.147,Y -512.291,Z 1270.781,A 0.000,B 0.000,C 90.000,E1 356.502} C_DIS
LIN {X 0.230,Y -515.604,Z 1270.777,A 0.000,B 0.000,C 90.000,E1 355.869} C_DIS
LIN {X -0.172,Y -519.399,Z 1270.773,A 0.000,B 0.000,C 90.000,E1 355.179} C_DIS
LIN {X -0.025,Y -522.919,Z 1270.769,A 0.000,B 0.000,C 90.000,E1 354.432} C_DIS
LIN {X 0.165,Y -527.503,Z 1270.763,A 0.000,B 0.000,C 90.000,E1 353.394} C_DIS
LIN {X -0.119,Y -531.498,Z 1270.758,A 0.000,B 0.000,C 90.000,E1 352.413} C_DIS
LIN {X -0.082,Y -534.664,Z 1270.753,A 0.000,B 0.000,C 90.000,E1 351.546} C_DIS
LIN {X -0.013,Y -537.514,Z 1270.748,A 0.000,B 0.000,C 90.000,E1 350.679} C_DIS
LIN {X 0.177,Y -540.091,Z 1270.744,A 0.000,B 0.000,C 90.000,E1 349.803} C_DIS
LIN {X -0.158,Y -543.258,Z 1270.737,A 0.000,B 0.000,C 90.000,E1 348.701} C_DIS
LIN {X 0.093,Y -545.293,Z 1270.732,A 0.000,B 0.000,C 90.000,E1 347.825} C_DIS
LIN {X 0.053,Y -547.801,Z 1270.726,A 0.000,B 0.000,C 90.000,E1 346.700} C_DIS
LIN {X -0.180,Y -549.436,Z 1270.722,A 0.000,B 0.000,C 90.000,E1 345.880} C_DIS
LIN {X -0.158,Y -551.404,Z 1270.715,A 0.000,B 0.000,C 90.000,E1 344.755} C_DIS
LIN {X 0.154,Y -553.343,Z 1270.708,A 0.000,B 0.000,C 90.000,E1 343.323} C_DIS
LIN {X -0.138,Y -554.543,Z 1270.701,A 0.000,B 0.000,C 90.000,E1 342.236} C_DIS
LIN {X -0.169,Y -555.147,Z 1270.697,A 0.000,B 0.000,C 90.000,E1 341.402} C_DIS
LIN {X -0.020,Y -555.486,Z 1270.692,A 0.000,B 0.000,C 90.000,E1 340.550} C_DIS
LIN {X -0.155,Y -555.541,Z 1270.689,A 0.000,B 0.000,C 90.000,E1 340.007} C_DIS
LIN {X -0.004,Y -555.304,Z 1270.684,A 0.000,B 0.000,C 90.000,E1 339.156} C_DIS
LIN {X -0.171,Y -554.747,Z 1270.680,A 0.000,B 0.000,C 90.000,E1 338.337} C_DIS
LIN {X -0.031,Y -553.960,Z 1270.675,A 0.000,B 0.000,C 90.000,E1 337.486} C_DIS
LIN {X 0.079,Y -552.271,Z 1270.669,A 0.000,B 0.000,C 90.000,E1 336.357} C_DIS
LIN {X 0.166,Y -550.251,Z 1270.662,A 0.000,B 0.000,C 90.000,E1 335.229} C_DIS
LIN {X -0.066,Y -549.735,Z 1270.661,A 0.000,B 0.000,C 90.000,E1 334.973} C_DIS
LIN {X 0.197,Y -549.018,Z 1270.659,A 0.000,B 0.000,C 90.000,E1 334.665} C_DIS
LIN {X -0.039,Y -548.481,Z 1270.658,A 0.000,B 0.000,C 90.000,E1 334.409} C_DIS
LIN {X 0.223,Y -545.456,Z 1270.652,A 0.000,B 0.000,C 90.000,E1 333.256} C_DIS
LIN {X 0.212,Y -542.756,Z 1270.647,A 0.000,B 0.000,C 90.000,E1 332.410} C_DIS
LIN {X -0.089,Y -538.432,Z 1270.641,A 0.000,B 0.000,C 90.000,E1 331.307} C_DIS
LIN {X -0.036,Y -535.177,Z 1270.637,A 0.000,B 0.000,C 90.000,E1 330.589} C_DIS
LIN {X 0.125,Y -532.267,Z 1270.633,A 0.000,B 0.000,C 90.000,E1 329.999} C_DIS
LIN {X -0.041,Y -527.373,Z 1270.629,A 0.000,B 0.000,C 90.000,E1 329.154} C_DIS
LIN {X -0.103,Y -518.598,Z 1270.621,A 0.000,B 0.000,C 90.000,E1 327.709} C_DIS
LIN {X -0.324,Y -512.423,Z 1270.615,A 0.000,B 0.000,C 90.000,E1 326.707} C_DIS
LIN {X -0.200,Y -508.340,Z 1270.610,A 0.000,B 0.000,C 90.000,E1 325.881} C_DIS
LIN {X 0.221,Y -506.313,Z 1270.608,A 0.000,B 0.000,C 90.000,E1 325.388} C_DIS
LIN {X -0.178,Y -503.866,Z 1270.604,A 0.000,B 0.000,C 90.000,E1 324.689} C_DIS
LIN {X 0.012,Y -502.449,Z 1270.600,A 0.000,B 0.000,C 90.000,E1 324.069} C_DIS
LIN {X -0.215,Y -501.341,Z 1270.597,A 0.000,B 0.000,C 90.000,E1 323.497} C_DIS
LIN {X 0.251,Y -500.637,Z 1270.594,A 0.000,B 0.000,C 90.000,E1 322.844} C_DIS
LIN {X -0.113,Y -500.046,Z 1270.589,A 0.000,B 0.000,C 90.000,E1 321.984} C_DIS
LIN {X 0.277,Y -499.749,Z 1270.580,A 0.000,B 0.000,C 90.000,E1 320.436} C_DIS
LIN {X -0.024,Y -500.038,Z 1270.569,A 0.000,B 0.000,C 90.000,E1 318.366} C_DIS
LIN {X -0.020,Y -500.362,Z 1270.560,A 0.000,B 0.000,C 90.000,E1 316.863} C_DIS
LIN {X -0.048,Y -500.600,Z 1270.552,A 0.000,B 0.000,C 90.000,E1 315.364} C_DIS
LIN {X -0.071,Y -500.925,Z 1270.544,A 0.000,B 0.000,C 90.000,E1 313.866} C_DIS
LIN {X -0.008,Y -501.344,Z 1270.532,A 0.000,B 0.000,C 90.000,E1 311.757} C_DIS
LIN {X -0.053,Y -501.544,Z 1270.527,A 0.000,B 0.000,C 90.000,E1 310.862} C_DIS
LIN {X -0.052,Y -501.806,Z 1270.514,A 0.000,B 0.000,C 90.000,E1 308.463} C_DIS
LIN {X -0.046,Y -502.143,Z 1270.504,A 0.000,B 0.000,C 90.000,E1 306.664} C_DIS
LIN {X 0.191,Y -502.318,Z 1270.497,A 0.000,B 0.000,C 90.000,E1 305.438} C_DIS
LIN {X -0.266,Y -502.388,Z 1270.489,A 0.000,B 0.000,C 90.000,E1 303.992} C_DIS
LIN {X -0.027,Y -502.217,Z 1270.480,A 0.000,B 0.000,C 90.000,E1 302.467} C_DIS
LIN {X 0.058,Y -502.112,Z 1270.474,A 0.000,B 0.000,C 90.000,E1 301.258} C_DIS
LIN {X -0.110,Y -501.815,Z 1270.467,A 0.000,B 0.000,C 90.000,E1 300.079} C_DIS
LIN {X -0.035,Y -501.255,Z 1270.460,A 0.000,B 0.000,C 90.000,E1 298.871} C_DIS
LIN {X -0.069,Y -500.434,Z 1270.455,A 0.000,B 0.000,C 90.000,E1 297.975} C_DIS
LIN {X -0.164,Y -499.676,Z 1270.452,A 0.000,B 0.000,C 90.000,E1 297.385} C_DIS
LIN {X 0.178,Y -498.647,Z 1270.449,A 0.000,B 0.000,C 90.000,E1 296.744} C_DIS
LIN {X -0.210,Y -497.995,Z 1270.447,A 0.000,B 0.000,C 90.000,E1 296.488} C_DIS
LIN {X 0.066,Y -497.161,Z 1270.445,A 0.000,B 0.000,C 90.000,E1 296.155} C_DIS
LIN {X 0.061,Y -490.969,Z 1270.437,A 0.000,B 0.000,C 90.000,E1 294.643} C_DIS
LIN {X -0.017,Y -478.704,Z 1270.418,A 0.000,B 0.000,C 90.000,E1 291.280} C_DIS
LIN {X -0.200,Y -468.492,Z 1270.399,A 0.000,B 0.000,C 90.000,E1 287.873} C_DIS
LIN {X -0.091,Y -459.592,Z 1270.378,A 0.000,B 0.000,C 90.000,E1 284.064} C_DIS
LIN {X 0.077,Y -452.053,Z 1270.353,A 0.000,B 0.000,C 90.000,E1 279.557} C_DIS
LIN {X -0.227,Y -446.554,Z 1270.319,A 0.000,B 0.000,C 90.000,E1 273.440} C_DIS
LIN {X -0.210,Y -449.686,Z 1270.259,A 0.000,B 0.000,C 90.000,E1 262.704} C_DIS
LIN {X 0.114,Y -456.486,Z 1270.233,A 0.000,B 0.000,C 90.000,E1 257.825} C_DIS
LIN {X 0.074,Y -465.201,Z 1270.209,A 0.000,B 0.000,C 90.000,E1 253.685} C_DIS
LIN {X 0.241,Y -470.976,Z 1270.197,A 0.000,B 0.000,C 90.000,E1 251.456} C_DIS
LIN {X 0.193,Y -471.558,Z 1270.195,A 0.000,B 0.000,C 90.000,E1 251.148} C_DIS
LIN {X -0.046,Y -472.275,Z 1270.192,A 0.000,B 0.000,C 90.000,E1 250.550} C_DIS
LIN {X -0.122,Y -472.658,Z 1270.188,A 0.000,B 0.000,C 90.000,E1 249.934} C_DIS
LIN {X 0.218,Y -472.882,Z 1270.183,A 0.000,B 0.000,C 90.000,E1 248.954} C_DIS
LIN {X 0.119,Y -472.943,Z 1270.178,A 0.000,B 0.000,C 90.000,E1 248.028} C_DIS
LIN {X -0.015,Y -472.450,Z 1270.171,A 0.000,B 0.000,C 90.000,E1 246.794} C_DIS
LIN {X -0.012,Y -471.555,Z 1270.162,A 0.000,B 0.000,C 90.000,E1 245.229} C_DIS
LIN {X 0.119,Y -470.348,Z 1270.152,A 0.000,B 0.000,C 90.000,E1 243.332} C_DIS
LIN {X 0.069,Y -469.422,Z 1270.143,A 0.000,B 0.000,C 90.000,E1 241.769} C_DIS
LIN {X 0.162,Y -468.381,Z 1270.133,A 0.000,B 0.000,C 90.000,E1 239.871} C_DIS
LIN {X -0.095,Y -467.377,Z 1270.124,A 0.000,B 0.000,C 90.000,E1 238.329} C_DIS
LIN {X -0.119,Y -466.167,Z 1270.115,A 0.000,B 0.000,C 90.000,E1 236.755} C_DIS
LIN {X -0.029,Y -464.887,Z 1270.105,A 0.000,B 0.000,C 90.000,E1 234.848} C_DIS
LIN {X 0.051,Y -464.009,Z 1270.096,A 0.000,B 0.000,C 90.000,E1 233.256} C_DIS
LIN {X -0.221,Y -462.635,Z 1270.080,A 0.000,B 0.000,C 90.000,E1 230.436} C_DIS
LIN {X 0.196,Y -461.824,Z 1270.068,A 0.000,B 0.000,C 90.000,E1 228.162} C_DIS
LIN {X -0.143,Y -461.231,Z 1270.057,A 0.000,B 0.000,C 90.000,E1 226.296} C_DIS
LIN {X 0.188,Y -460.583,Z 1270.045,A 0.000,B 0.000,C 90.000,E1 224.028} C_DIS
LIN {X 0.225,Y -460.567,Z 1270.020,A 0.000,B 0.000,C 90.000,E1 219.564} C_DIS
LIN {X -0.117,Y -461.691,Z 1270.002,A 0.000,B 0.000,C 90.000,E1 216.423} C_DIS
LIN {X 0.044,Y -464.429,Z 1269.983,A 0.000,B 0.000,C 90.000,E1 212.911} C_DIS
LIN {X 0.123,Y -466.512,Z 1269.972,A 0.000,B 0.000,C 90.000,E1 211.003} C_DIS
LIN {X -0.078,Y -469.179,Z 1269.960,A 0.000,B 0.000,C 90.000,E1 208.821} C_DIS
LIN {X -0.137,Y -470.947,Z 1269.951,A 0.000,B 0.000,C 90.000,E1 207.257} C_DIS
LIN {X 0.171,Y -473.814,Z 1269.939,A 0.000,B 0.000,C 90.000,E1 205.027} C_DIS
LIN {X -0.268,Y -477.092,Z 1269.927,A 0.000,B 0.000,C 90.000,E1 202.898} C_DIS
LIN {X 0.069,Y -482.240,Z 1269.910,A 0.000,B 0.000,C 90.000,E1 199.758} C_DIS
LIN {X -0.233,Y -485.592,Z 1269.900,A 0.000,B 0.000,C 90.000,E1 197.946} C_DIS
LIN {X 0.000,Y -489.143,Z 1269.889,A 0.000,B 0.000,C 90.000,E1 196.079} C_DIS
LIN {X -0.047,Y -493.850,Z 1269.876,A 0.000,B 0.000,C 90.000,E1 193.647} C_DIS
LIN {X -0.017,Y -497.555,Z 1269.866,A 0.000,B 0.000,C 90.000,E1 191.827} C_DIS
LIN {X 0.069,Y -500.628,Z 1269.857,A 0.000,B 0.000,C 90.000,E1 190.310} C_DIS
LIN {X 0.130,Y -503.706,Z 1269.849,A 0.000,B 0.000,C 90.000,E1 188.803} C_DIS
LIN {X 0.130,Y -507.541,Z 1269.839,A 0.000,B 0.000,C 90.000,E1 187.011} C_DIS
LIN {X 0.210,Y -511.233,Z 1269.829,A 0.000,B 0.000,C 90.000,E1 185.220} C_DIS
LIN {X -0.240,Y -514.892,Z 1269.819,A 0.000,B 0.000,C 90.000,E1 183.498} C_DIS
LIN {X -0.056,Y -517.828,Z 1269.811,A 0.000,B 0.000,C 90.000,E1 182.007} C_DIS
LIN {X 0.237,Y -520.071,Z 1269.805,A 0.000,B 0.000,C 90.000,E1 180.802} C_DIS
LIN {X -0.060,Y -523.352,Z 1269.795,A 0.000,B 0.000,C 90.000,E1 179.083} C_DIS
LIN {X -0.209,Y -525.498,Z 1269.788,A 0.000,B 0.000,C 90.000,E1 177.936} C_DIS
LIN {X 0.174,Y -527.906,Z 1269.780,A 0.000,B 0.000,C 90.000,E1 176.445} C_DIS
LIN {X 0.090,Y -529.641,Z 1269.774,A 0.000,B 0.000,C 90.000,E1 175.298} C_DIS
LIN {X 0.071,Y -531.235,Z 1269.768,A 0.000,B 0.000,C 90.000,E1 174.147} C_DIS
LIN {X 0.073,Y -532.558,Z 1269.761,A 0.000,B 0.000,C 90.000,E1 172.996} C_DIS
LIN {X 0.205,Y -533.945,Z 1269.753,A 0.000,B 0.000,C 90.000,E1 171.546} C_DIS
LIN {X -0.210,Y -534.931,Z 1269.747,A 0.000,B 0.000,C 90.000,E1 170.443} C_DIS
LIN {X -0.090,Y -535.630,Z 1269.740,A 0.000,B 0.000,C 90.000,E1 169.285} C_DIS
LIN {X 0.076,Y -536.022,Z 1269.736,A 0.000,B 0.000,C 90.000,E1 168.409} C_DIS
LIN {X -0.103,Y -536.360,Z 1269.729,A 0.000,B 0.000,C 90.000,E1 167.285} C_DIS
LIN {X -0.145,Y -536.649,Z 1269.720,A 0.000,B 0.000,C 90.000,E1 165.574} C_DIS
LIN {X -0.194,Y -537.053,Z 1269.710,A 0.000,B 0.000,C 90.000,E1 163.866} C_DIS
LIN {X 0.052,Y -537.806,Z 1269.701,A 0.000,B 0.000,C 90.000,E1 162.127} C_DIS
LIN {X -0.016,Y -539.515,Z 1269.691,A 0.000,B 0.000,C 90.000,E1 160.423} C_DIS
LIN {X -0.034,Y -540.878,Z 1269.687,A 0.000,B 0.000,C 90.000,E1 159.571} C_DIS
LIN {X 0.195,Y -543.483,Z 1269.680,A 0.000,B 0.000,C 90.000,E1 158.411} C_DIS
LIN {X -0.087,Y -546.116,Z 1269.676,A 0.000,B 0.000,C 90.000,E1 157.592} C_DIS
LIN {X -0.301,Y -548.185,Z 1269.672,A 0.000,B 0.000,C 90.000,E1 157.050} C_DIS
LIN {X -0.144,Y -552.359,Z 1269.667,A 0.000,B 0.000,C 90.000,E1 156.049} C_DIS
LIN {X -0.099,Y -555.297,Z 1269.664,A 0.000,B 0.000,C 90.000,E1 155.485} C_DIS
LIN {X 0.054,Y -562.078,Z 1269.658,A 0.000,B 0.000,C 90.000,E1 154.357} C_DIS
LIN {X 0.320,Y -566.743,Z 1269.654,A 0.000,B 0.000,C 90.000,E1 153.640} C_DIS
LIN {X -0.129,Y -571.619,Z 1269.650,A 0.000,B 0.000,C 90.000,E1 152.999} C_DIS
LIN {X 0.084,Y -578.915,Z 1269.645,A 0.000,B 0.000,C 90.000,E1 152.025} C_DIS
LIN {X -0.184,Y -587.017,Z 1269.639,A 0.000,B 0.000,C 90.000,E1 150.973} C_DIS
LIN {X 0.151,Y -589.930,Z 1269.636,A 0.000,B 0.000,C 90.000,E1 150.539} C_DIS
LIN {X 0.122,Y -595.960,Z 1269.632,A 0.000,B 0.000,C 90.000,E1 149.744} C_DIS
LIN {X -0.337,Y -602.418,Z 1269.627,A 0.000,B 0.000,C 90.000,E1 148.869} C_DIS
LIN {X 0.220,Y -610.373,Z 1269.620,A 0.000,B 0.000,C 90.000,E1 147.661} C_DIS
LIN {X -0.097,Y -614.525,Z 1269.617,A 0.000,B 0.000,C 90.000,E1 147.041} C_DIS
LIN {X -0.087,Y -620.732,Z 1269.611,A 0.000,B 0.000,C 90.000,E1 146.008} C_DIS
LIN {X 0.025,Y -624.943,Z 1269.607,A 0.000,B 0.000,C 90.000,E1 145.229} C_DIS
LIN {X 0.179,Y -629.470,Z 1269.602,A 0.000,B 0.000,C 90.000,E1 144.322} C_DIS
LIN {X 0.380,Y -633.655,Z 1269.597,A 0.000,B 0.000,C 90.000,E1 143.417} C_DIS
LIN {X 0.112,Y -637.819,Z 1269.591,A 0.000,B 0.000,C 90.000,E1 142.431} C_DIS
LIN {X 0.180,Y -642.567,Z 1269.584,A 0.000,B 0.000,C 90.000,E1 141.170} C_DIS
LIN {X 0.333,Y -646.758,Z 1269.578,A 0.000,B 0.000,C 90.000,E1 139.908} C_DIS
LIN {X 0.062,Y -650.572,Z 1269.571,A 0.000,B 0.000,C 90.000,E1 138.690} C_DIS
LIN {X -0.104,Y -653.616,Z 1269.565,A 0.000,B 0.000,C 90.000,E1 137.715} C_DIS
LIN {X 0.205,Y -656.430,Z 1269.560,A 0.000,B 0.000,C 90.000,E1 136.701} C_DIS
LIN {X -0.008,Y -662.154,Z 1269.549,A 0.000,B 0.000,C 90.000,E1 134.757} C_DIS
LIN {X -0.067,Y -665.881,Z 1269.542,A 0.000,B 0.000,C 90.000,E1 133.542} C_DIS
LIN {X -0.029,Y -670.333,Z 1269.534,A 0.000,B 0.000,C 90.000,E1 132.081} C_DIS
LIN {X 0.084,Y -673.917,Z 1269.527,A 0.000,B 0.000,C 90.000,E1 130.862} C_DIS
LIN {X 0.254,Y -677.435,Z 1269.520,A 0.000,B 0.000,C 90.000,E1 129.644} C_DIS
LIN {X 0.042,Y -680.790,Z 1269.514,A 0.000,B 0.000,C 90.000,E1 128.463} C_DIS
LIN {X -0.153,Y -683.396,Z 1269.508,A 0.000,B 0.000,C 90.000,E1 127.523} C_DIS
LIN {X -0.316,Y -685.904,Z 1269.503,A 0.000,B 0.000,C 90.000,E1 126.583} C_DIS
LIN {X 0.328,Y -689.339,Z 1269.495,A 0.000,B 0.000,C 90.000,E1 125.105} C_DIS
LIN {X -0.164,Y -691.514,Z 1269.490,A 0.000,B 0.000,C 90.000,E1 124.199} C_DIS
LIN {X -0.032,Y -693.920,Z 1269.483,A 0.000,B 0.000,C 90.000,E1 123.007} C_DIS
LIN {X 0.341,Y -696.212,Z 1269.477,A 0.000,B 0.000,C 90.000,E1 121.799} C_DIS
LIN {X -0.200,Y -698.337,Z 1269.470,A 0.000,B 0.000,C 90.000,E1 120.669} C_DIS
LIN {X -0.101,Y -700.460,Z 1269.463,A 0.000,B 0.000,C 90.000,E1 119.255} C_DIS
LIN {X -0.243,Y -701.399,Z 1269.459,A 0.000,B 0.000,C 90.000,E1 118.565} C_DIS
LIN {X 0.245,Y -702.503,Z 1269.453,A 0.000,B 0.000,C 90.000,E1 117.590} C_DIS
LIN {X -0.166,Y -703.030,Z 1269.450,A 0.000,B 0.000,C 90.000,E1 116.924} C_DIS
LIN {X -0.264,Y -703.266,Z 1269.446,A 0.000,B 0.000,C 90.000,E1 116.232} C_DIS
LIN {X 0.301,Y -703.290,Z 1269.443,A 0.000,B 0.000,C 90.000,E1 115.720} C_DIS
LIN {X -0.071,Y -703.119,Z 1269.440,A 0.000,B 0.000,C 90.000,E1 115.283} C_DIS
LIN {X -0.160,Y -702.498,Z 1269.437,A 0.000,B 0.000,C 90.000,E1 114.591} C_DIS
LIN {X -0.242,Y -701.766,Z 1269.434,A 0.000,B 0.000,C 90.000,E1 114.131} C_DIS
LIN {X 0.021,Y -700.054,Z 1269.431,A 0.000,B 0.000,C 90.000,E1 113.643} C_DIS
LIN {X 0.291,Y -699.040,Z 1269.430,A 0.000,B 0.000,C 90.000,E1 113.387} C_DIS
LIN {X 0.148,Y -698.173,Z 1269.429,A 0.000,B 0.000,C 90.000,E1 113.281} C_DIS
LIN {X 0.137,Y -694.196,Z 1269.427,A 0.000,B 0.000,C 90.000,E1 112.823} C_DIS
LIN {X -0.006,Y -692.714,Z 1269.426,A 0.000,B 0.000,C 90.000,E1 112.717} C_DIS
LIN {X 0.262,Y -690.589,Z 1269.426,A 0.000,B 0.000,C 90.000,E1 112.589} C_DIS
LIN {X -0.107,Y -688.093,Z 1269.425,A 0.000,B 0.000,C 90.000,E1 112.514} C_DIS
LIN {X -0.289,Y -681.993,Z 1269.424,A 0.000,B 0.000,C 90.000,E1 112.333} C_DIS
LIN {X 0.053,Y -677.635,Z 1269.423,A 0.000,B 0.000,C 90.000,E1 112.206} C_DIS
LIN {X 0.003,Y -669.972,Z 1269.423,A 0.000,B 0.000,C 90.000,E1 112.153} C_DIS
LIN {X -0.034,Y -635.510,Z 1269.423,A 0.000,B 0.000,C 90.000,E1 112.153} C_DIS
LIN {X 0.318,Y -632.086,Z 1269.423,A 0.000,B 0.000,C 90.000,E1 112.025} C_DIS
LIN {X 0.284,Y -632.059,Z 1269.423,A 0.000,B 0.000,C 90.000,E1 112.025} C_DIS
LIN {X 0.038,Y -631.889,Z 1269.422,A 0.000,B 0.000,C 90.000,E1 112.025} C_DIS
LIN {X -0.005,Y -631.860,Z 1269.422,A 0.000,B 0.000,C 90.000,E1 112.025} C_DIS
LIN {X -0.017,Y -632.205,Z 1269.421,A 0.000,B 0.000,C 90.000,E1 111.844} C_DIS
LIN {X -0.077,Y -635.025,Z 1269.419,A 0.000,B 0.000,C 90.000,E1 111.334} C_DIS
LIN {X 0.194,Y -641.137,Z 1269.414,A 0.000,B 0.000,C 90.000,E1 110.429} C_DIS
LIN {X 0.139,Y -645.200,Z 1269.410,A 0.000,B 0.000,C 90.000,E1 109.812} C_DIS
LIN {X -0.145,Y -648.669,Z 1269.407,A 0.000,B 0.000,C 90.000,E1 109.214} C_DIS
LIN {X -0.188,Y -651.869,Z 1269.403,A 0.000,B 0.000,C 90.000,E1 108.598} C_DIS
LIN {X 0.207,Y -654.897,Z 1269.400,A 0.000,B 0.000,C 90.000,E1 107.946} C_DIS
LIN {X 0.045,Y -658.277,Z 1269.396,A 0.000,B 0.000,C 90.000,E1 107.221} C_DIS
LIN {X -0.089,Y -661.380,Z 1269.392,A 0.000,B 0.000,C 90.000,E1 106.496} C_DIS
LIN {X -0.380,Y -664.108,Z 1269.388,A 0.000,B 0.000,C 90.000,E1 105.788} C_DIS
LIN {X 0.260,Y -665.675,Z 1269.385,A 0.000,B 0.000,C 90.000,E1 105.245} C_DIS
LIN {X 0.013,Y -667.641,Z 1269.381,A 0.000,B 0.000,C 90.000,E1 104.537} C_DIS
LIN {X -0.214,Y -669.058,Z 1269.377,A 0.000,B 0.000,C 90.000,E1 103.828} C_DIS
LIN {X 0.293,Y -669.796,Z 1269.374,A 0.000,B 0.000,C 90.000,E1 103.300} C_DIS
LIN {X 0.155,Y -670.259,Z 1269.371,A 0.000,B 0.000,C 90.000,E1 102.827} C_DIS
LIN {X -0.052,Y -670.615,Z 1269.367,A 0.000,B 0.000,C 90.000,E1 102.119} C_DIS
LIN {X -0.326,Y -670.537,Z 1269.365,A 0.000,B 0.000,C 90.000,E1 101.658} C_DIS
LIN {X 0.123,Y -670.009,Z 1269.361,A 0.000,B 0.000,C 90.000,E1 100.894} C_DIS
LIN {X -0.218,Y -669.019,Z 1269.357,A 0.000,B 0.000,C 90.000,E1 100.197} C_DIS
LIN {X -0.294,Y -668.600,Z 1269.355,A 0.000,B 0.000,C 90.000,E1 99.962} C_DIS
LIN {X 0.093,Y -667.477,Z 1269.353,A 0.000,B 0.000,C 90.000,E1 99.443} C_DIS
LIN {X -0.076,Y -666.004,Z 1269.350,A 0.000,B 0.000,C 90.000,E1 98.973} C_DIS
LIN {X -0.268,Y -665.170,Z 1269.349,A 0.000,B 0.000,C 90.000,E1 98.746} C_DIS
LIN {X 0.200,Y -663.216,Z 1269.346,A 0.000,B 0.000,C 90.000,E1 98.219} C_DIS
LIN {X -0.198,Y -660.301,Z 1269.342,A 0.000,B 0.000,C 90.000,E1 97.644} C_DIS
LIN {X 0.140,Y -657.624,Z 1269.340,A 0.000,B 0.000,C 90.000,E1 97.125} C_DIS
LIN {X -0.222,Y -653.776,Z 1269.336,A 0.000,B 0.000,C 90.000,E1 96.543} C_DIS
LIN {X -0.002,Y -650.298,Z 1269.333,A 0.000,B 0.000,C 90.000,E1 96.030} C_DIS
LIN {X 0.212,Y -645.423,Z 1269.330,A 0.000,B 0.000,C 90.000,E1 95.391} C_DIS
LIN {X -0.256,Y -641.090,Z 1269.327,A 0.000,B 0.000,C 90.000,E1 94.935} C_DIS
LIN {X -0.055,Y -636.363,Z 1269.325,A 0.000,B 0.000,C 90.000,E1 94.416} C_DIS
LIN {X 0.248,Y -630.181,Z 1269.321,A 0.000,B 0.000,C 90.000,E1 93.784} C_DIS
